LIN {X 0,Y 584.053,Z 357.982,A -85,B 0,C 180,E1 1855.602,E2 1855.602} C_VEL
LIN {X 0,Y 584.048,Z 357.978,A -85,B 0,C 180,E1 1852.272,E2 1852.272} C_VEL
LIN {X 0,Y 584.06,Z 357.981,A -85,B 0,C 180,E1 1849.289,E2 1849.289} C_VEL
LIN {X 0,Y 584.043,Z 357.976,A -85,B 0,C 180,E1 1845.968,E2 1845.968} C_VEL
LIN {X 0,Y 584.074,Z 357.982,A -85,B 0,C 180,E1 1842.948,E2 1842.948} C_VEL
LIN {X 0,Y 584.041,Z 357.978,A -85,B 0,C 180,E1 1839.765,E2 1839.765} C_VEL
LIN {X 0,Y 584.079,Z 357.983,A -85,B 0,C 180,E1 1836.687,E2 1836.687} C_VEL
LIN {X 0,Y 584.036,Z 357.983,A -85,B 0,C 180,E1 1833.454,E2 1833.454} C_VEL
LIN {X 0,Y 584.046,Z 358.076,A -85,B 0,C 180,E1 1833.218,E2 1833.218} C_VEL
LIN {X 0,Y 586.664,Z 365.487,A -85,B 0,C 180,E1 1832.47,E2 1832.47} C_VEL
LIN {X 0,Y 586.133,Z 402.245,A -85,B 0,C 180,E1 1829.65,E2 1829.65} C_VEL
LIN {X 0,Y 585.6,Z 444.184,A -85,B 0,C 180,E1 1826.531,E2 1826.531} C_VEL
LIN {X 0,Y 585.211,Z 489.388,A -85,B 0,C 180,E1 1823.299,E2 1823.299} C_VEL
LIN {X 0,Y 584.881,Z 536.224,A -85,B 0,C 180,E1 1820.024,E2 1820.024} C_VEL
LIN {X 0,Y 584.586,Z 583.959,A -85,B 0,C 180,E1 1816.75,E2 1816.75} C_VEL
LIN {X 0,Y 584.606,Z 588.885,A -85,B 0,C 180,E1 1816.44,E2 1816.44} C_VEL
LIN {X 0,Y 584.631,Z 729.653,A -85,B 0,C 180,E1 1814.662,E2 1814.662} C_VEL
LIN {X 0,Y 584.569,Z 745.603,A -85,B 0,C 180,E1 1814.307,E2 1814.307} C_VEL
LIN {X 0,Y 584.491,Z 761.576,A -85,B 0,C 180,E1 1813.756,E2 1813.756} C_VEL
LIN {X 0,Y 584.386,Z 776.468,A -85,B 0,C 180,E1 1813.053,E2 1813.053} C_VEL
LIN {X 0,Y 584.267,Z 791.891,A -85,B 0,C 180,E1 1812.094,E2 1812.094} C_VEL
LIN {X 0,Y 584.171,Z 804.549,A -85,B 0,C 180,E1 1811.093,E2 1811.093} C_VEL
LIN {X 0,Y 584.08,Z 817.071,A -85,B 0,C 180,E1 1809.857,E2 1809.857} C_VEL
LIN {X 0,Y 584.007,Z 827.449,A -85,B 0,C 180,E1 1808.566,E2 1808.566} C_VEL
LIN {X 0,Y 583.964,Z 836.343,A -85,B 0,C 180,E1 1807.18,E2 1807.18} C_VEL
LIN {X 0,Y 583.934,Z 843.646,A -85,B 0,C 180,E1 1805.7,E2 1805.7} C_VEL
LIN {X 0,Y 583.92,Z 849.058,A -85,B 0,C 180,E1 1804.223,E2 1804.223} C_VEL
LIN {X 0,Y 583.917,Z 852.97,A -85,B 0,C 180,E1 1802.65,E2 1802.65} C_VEL
LIN {X 0,Y 583.916,Z 855.029,A -85,B 0,C 180,E1 1801.08,E2 1801.08} C_VEL
LIN {X 0,Y 583.915,Z 855.387,A -85,B 0,C 180,E1 1799.412,E2 1799.412} C_VEL
LIN {X 0,Y 583.917,Z 853.911,A -85,B 0,C 180,E1 1797.841,E2 1797.841} C_VEL
LIN {X 0,Y 583.917,Z 850.708,A -85,B 0,C 180,E1 1796.269,E2 1796.269} C_VEL
LIN {X 0,Y 583.93,Z 845.646,A -85,B 0,C 180,E1 1794.695,E2 1794.695} C_VEL
LIN {X 0,Y 583.951,Z 838.942,A -85,B 0,C 180,E1 1793.215,E2 1793.215} C_VEL
LIN {X 0,Y 583.99,Z 830.831,A -85,B 0,C 180,E1 1791.831,E2 1791.831} C_VEL
LIN {X 0,Y 584.047,Z 821.249,A -85,B 0,C 180,E1 1790.541,E2 1790.541} C_VEL
LIN {X 0,Y 584.123,Z 810.24,A -85,B 0,C 180,E1 1789.347,E2 1789.347} C_VEL
LIN {X 0,Y 584.227,Z 797.718,A -85,B 0,C 180,E1 1788.249,E2 1788.249} C_VEL
LIN {X 0,Y 584.311,Z 784.011,A -85,B 0,C 180,E1 1787.298,E2 1787.298} C_VEL
LIN {X 0,Y 584.435,Z 769.379,A -85,B 0,C 180,E1 1786.496,E2 1786.496} C_VEL
LIN {X 0,Y 584.531,Z 754.061,A -85,B 0,C 180,E1 1785.872,E2 1785.872} C_VEL
LIN {X 0,Y 584.589,Z 738.598,A -85,B 0,C 180,E1 1785.426,E2 1785.426} C_VEL
LIN {X 0,Y 584.658,Z 721.58,A -85,B 0,C 180,E1 1785.13,E2 1785.13} C_VEL
LIN {X 0,Y 584.618,Z 588.986,A -85,B 0,C 180,E1 1783.472,E2 1783.472} C_VEL
LIN {X 0,Y 584.737,Z 556.999,A -85,B 0,C 180,E1 1781.317,E2 1781.317} C_VEL
LIN {X 0,Y 585.048,Z 511.693,A -85,B 0,C 180,E1 1778.179,E2 1778.179} C_VEL
LIN {X 0,Y 585.395,Z 465.881,A -85,B 0,C 180,E1 1774.939,E2 1774.939} C_VEL
LIN {X 0,Y 585.703,Z 443.805,A -85,B 0,C 180,E1 1773.323,E2 1773.323} C_VEL
LIN {X 0,Y 588.407,Z 405.449,A -85,B 0,C 180,E1 1770.07,E2 1770.07} C_VEL
LIN {X 0,Y 590.186,Z 385.24,A -85,B 0,C 180,E1 1768.262,E2 1768.262} C_VEL
LIN {X 0,Y 590.783,Z 371.274,A -85,B 0,C 180,E1 1766.805,E2 1766.805} C_VEL
LIN {X 0,Y 589.039,Z 367.53,A -85,B 0,C 180,E1 1766.051,E2 1766.051} C_VEL
LIN {X 0,Y 587.248,Z 364.067,A -85,B 0,C 180,E1 1765.224,E2 1765.224} C_VEL
LIN {X 0,Y 586.619,Z 362.881,A -85,B 0,C 180,E1 1764.899,E2 1764.899} C_VEL
LIN {X 0,Y 584.541,Z 359.787,A -85,B 0,C 180,E1 1763.673,E2 1763.673} C_VEL
LIN {X 0,Y 584.088,Z 358.254,A -85,B 0,C 180,E1 1762.7,E2 1762.7} C_VEL
LIN {X 0,Y 584.246,Z 358.829,A -85,B 0,C 180,E1 1761.928,E2 1761.928} C_VEL
LIN {X 0,Y 585.191,Z 361.195,A -85,B 0,C 180,E1 1761.167,E2 1761.167} C_VEL
LIN {X 0,Y 586.92,Z 363.366,A -85,B 0,C 180,E1 1760.612,E2 1760.612} C_VEL
LIN {X 0,Y 588.669,Z 367.246,A -85,B 0,C 180,E1 1760.057,E2 1760.057} C_VEL
LIN {X 0,Y 587.26,Z 390.715,A -85,B 0,C 180,E1 1758.655,E2 1758.655} C_VEL
LIN {X 0,Y 586.847,Z 427.382,A -85,B 0,C 180,E1 1756.679,E2 1756.679} C_VEL
LIN {X 0,Y 588.252,Z 442.511,A -85,B 0,C 180,E1 1755.823,E2 1755.823} C_VEL
LIN {X 0,Y 590.921,Z 453.438,A -85,B 0,C 180,E1 1755.124,E2 1755.124} C_VEL
LIN {X 0,Y 593.407,Z 459.109,A -85,B 0,C 180,E1 1754.68,E2 1754.68} C_VEL
LIN {X 0,Y 595.801,Z 462.899,A -85,B 0,C 180,E1 1754.227,E2 1754.227} C_VEL
LIN {X 0,Y 597.93,Z 465.232,A -85,B 0,C 180,E1 1753.748,E2 1753.748} C_VEL
LIN {X 0,Y 599.643,Z 466.302,A -85,B 0,C 180,E1 1753.226,E2 1753.226} C_VEL
LIN {X 0,Y 600.735,Z 465.901,A -85,B 0,C 180,E1 1752.637,E2 1752.637} C_VEL
LIN {X 0,Y 600.838,Z 464.09,A -85,B 0,C 180,E1 1752.117,E2 1752.117} C_VEL
LIN {X 0,Y 599.969,Z 460.825,A -85,B 0,C 180,E1 1751.63,E2 1751.63} C_VEL
LIN {X 0,Y 598.197,Z 456.293,A -85,B 0,C 180,E1 1751.238,E2 1751.238} C_VEL
LIN {X 0,Y 595.49,Z 449.308,A -85,B 0,C 180,E1 1750.915,E2 1750.915} C_VEL
LIN {X 0,Y 593.429,Z 440.344,A -85,B 0,C 180,E1 1750.685,E2 1750.685} C_VEL
LIN {X 0,Y 592.253,Z 428.653,A -85,B 0,C 180,E1 1750.553,E2 1750.553} C_VEL
LIN {X 0,Y 592.038,Z 404.531,A -85,B 0,C 180,E1 1750.528,E2 1750.528} C_VEL
LIN {X 0,Y 592.025,Z 368.885,A -85,B 0,C 180,E1 1750.527,E2 1750.527} C_VEL
LIN {X 0,Y 589.112,Z 365.245,A -85,B 0,C 180,E1 1750.194,E2 1750.194} C_VEL
LIN {X 0,Y 588.306,Z 364.085,A -85,B 0,C 180,E1 1750.101,E2 1750.101} C_VEL
LIN {X 0,Y 585.578,Z 361.73,A -85,B 0,C 180,E1 1749.783,E2 1749.783} C_VEL
LIN {X 0,Y 584.22,Z 358.714,A -85,B 0,C 180,E1 1749.623,E2 1749.623} C_VEL
LIN {X 0,Y 584.097,Z 357.981,A -85,B 0,C 180,E1 1749.585,E2 1749.585} C_VEL
LIN {X 0,Y 584.102,Z 357.996,A -85,B 0,C 180,E1 1749.495,E2 1749.495} C_VEL
LIN {X 0,Y 585.487,Z 361.592,A -85,B 0,C 180,E1 1749.167,E2 1749.167} C_VEL
LIN {X 0,Y 587.967,Z 367.026,A -85,B 0,C 180,E1 1748.647,E2 1748.647} C_VEL
LIN {X 0,Y 587.4,Z 418.925,A -85,B 0,C 180,E1 1745.668,E2 1745.668} C_VEL
LIN {X 0,Y 587.163,Z 455.345,A -85,B 0,C 180,E1 1743.661,E2 1743.661} C_VEL
LIN {X 0,Y 587.671,Z 460.738,A -85,B 0,C 180,E1 1743.55,E2 1743.55} C_VEL
LIN {X 0,Y 587.067,Z 677.552,A -85,B 0,C 180,E1 1740.523,E2 1740.523} C_VEL
LIN {X 0,Y 586.8,Z 761.949,A -85,B 0,C 180,E1 1739.34,E2 1739.34} C_VEL
LIN {X 0,Y 586.619,Z 783.698,A -85,B 0,C 180,E1 1738.843,E2 1738.843} C_VEL
LIN {X 0,Y 586.357,Z 806.115,A -85,B 0,C 180,E1 1738.137,E2 1738.137} C_VEL
LIN {X 0,Y 586.113,Z 827.151,A -85,B 0,C 180,E1 1737.28,E2 1737.28} C_VEL
LIN {X 0,Y 585.823,Z 846.743,A -85,B 0,C 180,E1 1736.29,E2 1736.29} C_VEL
LIN {X 0,Y 585.487,Z 867.144,A -85,B 0,C 180,E1 1735.057,E2 1735.057} C_VEL
LIN {X 0,Y 585.219,Z 885.801,A -85,B 0,C 180,E1 1733.726,E2 1733.726} C_VEL
LIN {X 0,Y 584.927,Z 904.1,A -85,B 0,C 180,E1 1732.196,E2 1732.196} C_VEL
LIN {X 0,Y 584.66,Z 921.221,A -85,B 0,C 180,E1 1730.523,E2 1730.523} C_VEL
LIN {X 0,Y 584.434,Z 936.724,A -85,B 0,C 180,E1 1728.762,E2 1728.762} C_VEL
LIN {X 0,Y 584.265,Z 950.748,A -85,B 0,C 180,E1 1726.914,E2 1726.914} C_VEL
LIN {X 0,Y 584.139,Z 963.342,A -85,B 0,C 180,E1 1724.979,E2 1724.979} C_VEL
LIN {X 0,Y 584.036,Z 974.372,A -85,B 0,C 180,E1 1722.96,E2 1722.96} C_VEL
LIN {X 0,Y 583.972,Z 983.482,A -85,B 0,C 180,E1 1720.956,E2 1720.956} C_VEL
LIN {X 0,Y 583.942,Z 991.15,A -85,B 0,C 180,E1 1718.897,E2 1718.897} C_VEL
LIN {X 0,Y 583.922,Z 997.17,A -85,B 0,C 180,E1 1716.786,E2 1716.786} C_VEL
LIN {X 0,Y 583.908,Z 1001.629,A -85,B 0,C 180,E1 1714.616,E2 1714.616} C_VEL
LIN {X 0,Y 583.897,Z 1004.326,A -85,B 0,C 180,E1 1712.552,E2 1712.552} C_VEL
LIN {X 0,Y 583.892,Z 1005.395,A -85,B 0,C 180,E1 1710.491,E2 1710.491} C_VEL
LIN {X 0,Y 583.899,Z 1004.954,A -85,B 0,C 180,E1 1708.332,E2 1708.332} C_VEL
LIN {X 0,Y 583.908,Z 1002.879,A -85,B 0,C 180,E1 1706.171,E2 1706.171} C_VEL
LIN {X 0,Y 583.918,Z 998.994,A -85,B 0,C 180,E1 1704.005,E2 1704.005} C_VEL
LIN {X 0,Y 583.937,Z 993.38,A -85,B 0,C 180,E1 1701.83,E2 1701.83} C_VEL
LIN {X 0,Y 583.97,Z 986.319,A -85,B 0,C 180,E1 1699.743,E2 1699.743} C_VEL
LIN {X 0,Y 584.013,Z 977.76,A -85,B 0,C 180,E1 1697.743,E2 1697.743} C_VEL
LIN {X 0,Y 584.102,Z 966.828,A -85,B 0,C 180,E1 1695.629,E2 1695.629} C_VEL
LIN {X 0,Y 584.228,Z 954.996,A -85,B 0,C 180,E1 1693.7,E2 1693.7} C_VEL
LIN {X 0,Y 584.377,Z 941.692,A -85,B 0,C 180,E1 1691.857,E2 1691.857} C_VEL
LIN {X 0,Y 584.559,Z 926.966,A -85,B 0,C 180,E1 1690.1,E2 1690.1} C_VEL
LIN {X 0,Y 584.807,Z 910.257,A -85,B 0,C 180,E1 1688.38,E2 1688.38} C_VEL
LIN {X 0,Y 585.104,Z 892.798,A -85,B 0,C 180,E1 1686.833,E2 1686.833} C_VEL
LIN {X 0,Y 585.409,Z 874.297,A -85,B 0,C 180,E1 1685.425,E2 1685.425} C_VEL
LIN {X 0,Y 585.679,Z 855.207,A -85,B 0,C 180,E1 1684.194,E2 1684.194} C_VEL
LIN {X 0,Y 585.986,Z 834.298,A -85,B 0,C 180,E1 1683.063,E2 1683.063} C_VEL
LIN {X 0,Y 586.307,Z 813.562,A -85,B 0,C 180,E1 1682.143,E2 1682.143} C_VEL
LIN {X 0,Y 586.515,Z 792.316,A -85,B 0,C 180,E1 1681.403,E2 1681.403} C_VEL
LIN {X 0,Y 586.726,Z 770.495,A -85,B 0,C 180,E1 1680.835,E2 1680.835} C_VEL
LIN {X 0,Y 586.869,Z 748.47,A -85,B 0,C 180,E1 1680.447,E2 1680.447} C_VEL
LIN {X 0,Y 587.486,Z 523.259,A -85,B 0,C 180,E1 1677.332,E2 1677.332} C_VEL
LIN {X 0,Y 587.485,Z 457.398,A -85,B 0,C 180,E1 1676.39,E2 1676.39} C_VEL
LIN {X 0,Y 587.058,Z 453.716,A -85,B 0,C 180,E1 1676.274,E2 1676.274} C_VEL
LIN {X 0,Y 587.62,Z 399.078,A -85,B 0,C 180,E1 1673.206,E2 1673.206} C_VEL
LIN {X 0,Y 587.877,Z 366.607,A -85,B 0,C 180,E1 1671.321,E2 1671.321} C_VEL
LIN {X 0,Y 584.335,Z 359.15,A -85,B 0,C 180,E1 1670.594,E2 1670.594} C_VEL
LIN {X 0,Y 584.1,Z 357.98,A -85,B 0,C 180,E1 1670.479,E2 1670.479} C_VEL
LIN {X 0,Y 584.117,Z 358.139,A -85,B 0,C 180,E1 1670.389,E2 1670.389} C_VEL
LIN {X 0,Y 585.254,Z 361.253,A -85,B 0,C 180,E1 1670.255,E2 1670.255} C_VEL
LIN {X 0,Y 587.659,Z 363.706,A -85,B 0,C 180,E1 1669.974,E2 1669.974} C_VEL
LIN {X 0,Y 588.786,Z 364.64,A -85,B 0,C 180,E1 1669.844,E2 1669.844} C_VEL
LIN {X 0,Y 591.535,Z 368.425,A -85,B 0,C 180,E1 1669.529,E2 1669.529} C_VEL
LIN {X 0,Y 592.035,Z 369.258,A -85,B 0,C 180,E1 1669.472,E2 1669.472} C_VEL
LIN {X 0,Y 592.224,Z 428.062,A -85,B 0,C 180,E1 1669.451,E2 1669.451} C_VEL
LIN {X 0,Y 593.343,Z 439.819,A -85,B 0,C 180,E1 1669.325,E2 1669.325} C_VEL
LIN {X 0,Y 595.364,Z 448.897,A -85,B 0,C 180,E1 1669.099,E2 1669.099} C_VEL
LIN {X 0,Y 598.058,Z 455.968,A -85,B 0,C 180,E1 1668.783,E2 1668.783} C_VEL
LIN {X 0,Y 599.889,Z 460.588,A -85,B 0,C 180,E1 1668.396,E2 1668.396} C_VEL
LIN {X 0,Y 600.807,Z 463.9,A -85,B 0,C 180,E1 1667.921,E2 1667.921} C_VEL
LIN {X 0,Y 600.841,Z 465.595,A -85,B 0,C 180,E1 1667.493,E2 1667.493} C_VEL
LIN {X 0,Y 600.174,Z 466.341,A -85,B 0,C 180,E1 1666.999,E2 1666.999} C_VEL
LIN {X 0,Y 598.675,Z 465.808,A -85,B 0,C 180,E1 1666.454,E2 1666.454} C_VEL
LIN {X 0,Y 596.53,Z 463.815,A -85,B 0,C 180,E1 1665.926,E2 1665.926} C_VEL
LIN {X 0,Y 593.903,Z 460.001,A -85,B 0,C 180,E1 1665.409,E2 1665.409} C_VEL
LIN {X 0,Y 591.267,Z 453.332,A -85,B 0,C 180,E1 1664.774,E2 1664.774} C_VEL
LIN {X 0,Y 589.42,Z 442.401,A -85,B 0,C 180,E1 1663.932,E2 1663.932} C_VEL
LIN {X 0,Y 589.031,Z 425.656,A -85,B 0,C 180,E1 1662.836,E2 1662.836} C_VEL
LIN {X 0,Y 589.555,Z 385.431,A -85,B 0,C 180,E1 1660.252,E2 1660.252} C_VEL
LIN {X 0,Y 589.749,Z 369.393,A -85,B 0,C 180,E1 1659.163,E2 1659.163} C_VEL
LIN {X 0,Y 586.078,Z 362.328,A -85,B 0,C 180,E1 1658.264,E2 1658.264} C_VEL
LIN {X 0,Y 584.273,Z 358.951,A -85,B 0,C 180,E1 1657.817,E2 1657.817} C_VEL
LIN {X 0,Y 584.093,Z 357.982,A -85,B 0,C 180,E1 1657.704,E2 1657.704} C_VEL
LIN {X 0,Y 584.07,Z 357.984,A -85,B 0,C 180,E1 1654.515,E2 1654.515} C_VEL
LIN {X 0,Y 584.087,Z 357.981,A -85,B 0,C 180,E1 1651.244,E2 1651.244} C_VEL
LIN {X 0,Y 584.097,Z 357.98,A -85,B 0,C 180,E1 1647.959,E2 1647.959} C_VEL
LIN {X 0,Y 584.087,Z 357.982,A -85,B 0,C 180,E1 1644.635,E2 1644.635} C_VEL
LIN {X 0,Y 584.1,Z 357.98,A -85,B 0,C 180,E1 1641.375,E2 1641.375} C_VEL
LIN {X 0,Y 584.098,Z 357.981,A -85,B 0,C 180,E1 1638.049,E2 1638.049} C_VEL
LIN {X 0,Y 584.092,Z 357.982,A -85,B 0,C 180,E1 1634.721,E2 1634.721} C_VEL
LIN {X 0,Y 584.1,Z 357.981,A -85,B 0,C 180,E1 1631.453,E2 1631.453} C_VEL
LIN {X 0,Y 584.092,Z 357.981,A -85,B 0,C 180,E1 1628.168,E2 1628.168} C_VEL
LIN {X 0,Y 584.084,Z 357.982,A -85,B 0,C 180,E1 1624.91,E2 1624.91} C_VEL
LIN {X 0,Y 584.095,Z 357.981,A -85,B 0,C 180,E1 1621.667,E2 1621.667} C_VEL
LIN {X 0,Y 584.084,Z 357.983,A -85,B 0,C 180,E1 1618.43,E2 1618.43} C_VEL
LIN {X 0,Y 584.099,Z 357.979,A -85,B 0,C 180,E1 1615.09,E2 1615.09} C_VEL
LIN {X 0,Y 584.079,Z 357.982,A -85,B 0,C 180,E1 1611.831,E2 1611.831} C_VEL
LIN {X 0,Y 584.092,Z 357.979,A -85,B 0,C 180,E1 1608.546,E2 1608.546} C_VEL
LIN {X 0,Y 584.096,Z 357.977,A -85,B 0,C 180,E1 1606.725,E2 1606.725} C_VEL
LIN {X 0,Y 583.11,Z 358.101,A -85,B 0,C 180,E1 1605.97,E2 1605.97} C_VEL
LIN {X 0,Y 576.657,Z 358.908,A -85,B 0,C 180,E1 1603.849,E2 1603.849} C_VEL
LIN {X 0,Y 576.112,Z 358.97,A -85,B 0,C 180,E1 1603.297,E2 1603.297} C_VEL
LIN {X 0,Y 576.132,Z 358.967,A -85,B 0,C 180,E1 1599.902,E2 1599.902} C_VEL
LIN {X 0,Y 576.129,Z 358.967,A -85,B 0,C 180,E1 1596.799,E2 1596.799} C_VEL
LIN {X 0,Y 576.111,Z 358.969,A -85,B 0,C 180,E1 1593.354,E2 1593.354} C_VEL
LIN {X 0,Y 576.151,Z 358.965,A -85,B 0,C 180,E1 1590.193,E2 1590.193} C_VEL
LIN {X 0,Y 576.105,Z 358.971,A -85,B 0,C 180,E1 1586.958,E2 1586.958} C_VEL
LIN {X 0,Y 576.154,Z 358.958,A -85,B 0,C 180,E1 1583.717,E2 1583.717} C_VEL
LIN {X 0,Y 576.109,Z 358.971,A -85,B 0,C 180,E1 1580.562,E2 1580.562} C_VEL
LIN {X 0,Y 576.137,Z 358.963,A -85,B 0,C 180,E1 1577.231,E2 1577.231} C_VEL
LIN {X 0,Y 576.126,Z 358.968,A -85,B 0,C 180,E1 1574.07,E2 1574.07} C_VEL
LIN {X 0,Y 576.115,Z 358.971,A -85,B 0,C 180,E1 1570.603,E2 1570.603} C_VEL
LIN {X 0,Y 576.151,Z 358.966,A -85,B 0,C 180,E1 1567.401,E2 1567.401} C_VEL
LIN {X 0,Y 576.105,Z 358.973,A -85,B 0,C 180,E1 1564.096,E2 1564.096} C_VEL
LIN {X 0,Y 576.174,Z 359.101,A -85,B 0,C 180,E1 1561.62,E2 1561.62} C_VEL
LIN {X 0,Y 578.943,Z 367.46,A -85,B 0,C 180,E1 1560.859,E2 1560.859} C_VEL
LIN {X 0,Y 578.406,Z 412.862,A -85,B 0,C 180,E1 1557.654,E2 1557.654} C_VEL
LIN {X 0,Y 577.861,Z 459.008,A -85,B 0,C 180,E1 1554.477,E2 1554.477} C_VEL
LIN {X 0,Y 577.806,Z 473.594,A -85,B 0,C 180,E1 1553.511,E2 1553.511} C_VEL
LIN {X 0,Y 578.38,Z 479.879,A -85,B 0,C 180,E1 1553.403,E2 1553.403} C_VEL
LIN {X 0,Y 577.837,Z 682.682,A -85,B 0,C 180,E1 1550.733,E2 1550.733} C_VEL
LIN {X 0,Y 577.692,Z 701.758,A -85,B 0,C 180,E1 1550.294,E2 1550.294} C_VEL
LIN {X 0,Y 577.499,Z 720.276,A -85,B 0,C 180,E1 1549.673,E2 1549.673} C_VEL
LIN {X 0,Y 577.252,Z 737.733,A -85,B 0,C 180,E1 1548.899,E2 1548.899} C_VEL
LIN {X 0,Y 577.042,Z 754.491,A -85,B 0,C 180,E1 1547.96,E2 1547.96} C_VEL
LIN {X 0,Y 576.794,Z 770.907,A -85,B 0,C 180,E1 1546.827,E2 1546.827} C_VEL
LIN {X 0,Y 576.56,Z 786.253,A -85,B 0,C 180,E1 1545.541,E2 1545.541} C_VEL
LIN {X 0,Y 576.357,Z 800.254,A -85,B 0,C 180,E1 1544.128,E2 1544.128} C_VEL
LIN {X 0,Y 576.205,Z 812.631,A -85,B 0,C 180,E1 1542.629,E2 1542.629} C_VEL
LIN {X 0,Y 576.087,Z 823.733,A -85,B 0,C 180,E1 1541.006,E2 1541.006} C_VEL
LIN {X 0,Y 575.998,Z 833.301,A -85,B 0,C 180,E1 1539.29,E2 1539.29} C_VEL
LIN {X 0,Y 575.956,Z 840.909,A -85,B 0,C 180,E1 1537.581,E2 1537.581} C_VEL
LIN {X 0,Y 575.92,Z 847.08,A -85,B 0,C 180,E1 1535.779,E2 1535.779} C_VEL
LIN {X 0,Y 575.919,Z 851.486,A -85,B 0,C 180,E1 1533.982,E2 1533.982} C_VEL
LIN {X 0,Y 575.917,Z 854.35,A -85,B 0,C 180,E1 1532.089,E2 1532.089} C_VEL
LIN {X 0,Y 575.911,Z 855.452,A -85,B 0,C 180,E1 1530.199,E2 1530.199} C_VEL
LIN {X 0,Y 575.913,Z 854.812,A -85,B 0,C 180,E1 1528.308,E2 1528.308} C_VEL
LIN {X 0,Y 575.909,Z 852.418,A -85,B 0,C 180,E1 1526.416,E2 1526.416} C_VEL
LIN {X 0,Y 575.923,Z 848.205,A -85,B 0,C 180,E1 1524.52,E2 1524.52} C_VEL
LIN {X 0,Y 575.941,Z 842.423,A -85,B 0,C 180,E1 1522.719,E2 1522.719} C_VEL
LIN {X 0,Y 575.998,Z 834.753,A -85,B 0,C 180,E1 1520.911,E2 1520.911} C_VEL
LIN {X 0,Y 576.07,Z 825.537,A -85,B 0,C 180,E1 1519.196,E2 1519.196} C_VEL
LIN {X 0,Y 576.188,Z 814.823,A -85,B 0,C 180,E1 1517.574,E2 1517.574} C_VEL
LIN {X 0,Y 576.334,Z 802.618,A -85,B 0,C 180,E1 1516.046,E2 1516.046} C_VEL
LIN {X 0,Y 576.522,Z 788.855,A -85,B 0,C 180,E1 1514.612,E2 1514.612} C_VEL
LIN {X 0,Y 576.747,Z 773.367,A -85,B 0,C 180,E1 1513.275,E2 1513.275} C_VEL
LIN {X 0,Y 576.986,Z 757.406,A -85,B 0,C 180,E1 1512.138,E2 1512.138} C_VEL
LIN {X 0,Y 577.194,Z 740.427,A -85,B 0,C 180,E1 1511.151,E2 1511.151} C_VEL
LIN {X 0,Y 577.461,Z 722.315,A -85,B 0,C 180,E1 1510.319,E2 1510.319} C_VEL
LIN {X 0,Y 577.664,Z 703.601,A -85,B 0,C 180,E1 1509.67,E2 1509.67} C_VEL
LIN {X 0,Y 577.822,Z 684.635,A -85,B 0,C 180,E1 1509.213,E2 1509.213} C_VEL
LIN {X 0,Y 577.938,Z 649.04,A -85,B 0,C 180,E1 1508.715,E2 1508.715} C_VEL
LIN {X 0,Y 578.207,Z 476.163,A -85,B 0,C 180,E1 1506.451,E2 1506.451} C_VEL
LIN {X 0,Y 577.737,Z 472.964,A -85,B 0,C 180,E1 1506.381,E2 1506.381} C_VEL
LIN {X 0,Y 578.229,Z 426.058,A -85,B 0,C 180,E1 1503.172,E2 1503.172} C_VEL
LIN {X 0,Y 578.809,Z 380.74,A -85,B 0,C 180,E1 1499.993,E2 1499.993} C_VEL
LIN {X 0,Y 578.729,Z 366.59,A -85,B 0,C 180,E1 1498.974,E2 1498.974} C_VEL
LIN {X 0,Y 576.1,Z 358.973,A -85,B 0,C 180,E1 1498.259,E2 1498.259} C_VEL
LIN {X 0,Y 576.155,Z 358.968,A -85,B 0,C 180,E1 1495.17,E2 1495.17} C_VEL
LIN {X 0,Y 576.096,Z 358.969,A -85,B 0,C 180,E1 1491.966,E2 1491.966} C_VEL
LIN {X 0,Y 576.163,Z 358.967,A -85,B 0,C 180,E1 1488.865,E2 1488.865} C_VEL
LIN {X 0,Y 576.096,Z 358.965,A -85,B 0,C 180,E1 1485.757,E2 1485.757} C_VEL
LIN {X 0,Y 576.16,Z 358.965,A -85,B 0,C 180,E1 1482.594,E2 1482.594} C_VEL
LIN {X 0,Y 576.095,Z 358.969,A -85,B 0,C 180,E1 1479.436,E2 1479.436} C_VEL
LIN {X 0,Y 576.157,Z 358.968,A -85,B 0,C 180,E1 1476.2,E2 1476.2} C_VEL
LIN {X 0,Y 576.127,Z 359.09,A -85,B 0,C 180,E1 1473.686,E2 1473.686} C_VEL
LIN {X 0,Y 579.582,Z 369.103,A -85,B 0,C 180,E1 1472.661,E2 1472.661} C_VEL
LIN {X 0,Y 579.005,Z 403.591,A -85,B 0,C 180,E1 1469.995,E2 1469.995} C_VEL
LIN {X 0,Y 578.244,Z 446.177,A -85,B 0,C 180,E1 1466.772,E2 1466.772} C_VEL
LIN {X 0,Y 577.665,Z 490.746,A -85,B 0,C 180,E1 1463.525,E2 1463.525} C_VEL
LIN {X 0,Y 577.219,Z 537.432,A -85,B 0,C 180,E1 1460.217,E2 1460.217} C_VEL
LIN {X 0,Y 576.827,Z 584.719,A -85,B 0,C 180,E1 1456.931,E2 1456.931} C_VEL
LIN {X 0,Y 576.855,Z 588.993,A -85,B 0,C 180,E1 1456.666,E2 1456.666} C_VEL
LIN {X 0,Y 577.147,Z 600.883,A -85,B 0,C 180,E1 1456.506,E2 1456.506} C_VEL
LIN {X 0,Y 576.881,Z 731.55,A -85,B 0,C 180,E1 1454.832,E2 1454.832} C_VEL
LIN {X 0,Y 576.789,Z 748.94,A -85,B 0,C 180,E1 1454.404,E2 1454.404} C_VEL
LIN {X 0,Y 576.665,Z 764.063,A -85,B 0,C 180,E1 1453.839,E2 1453.839} C_VEL
LIN {X 0,Y 576.528,Z 779.188,A -85,B 0,C 180,E1 1453.081,E2 1453.081} C_VEL
LIN {X 0,Y 576.379,Z 793.149,A -85,B 0,C 180,E1 1452.168,E2 1452.168} C_VEL
LIN {X 0,Y 576.252,Z 805.576,A -85,B 0,C 180,E1 1451.155,E2 1451.155} C_VEL
LIN {X 0,Y 576.127,Z 817.926,A -85,B 0,C 180,E1 1449.894,E2 1449.894} C_VEL
LIN {X 0,Y 576.042,Z 827.443,A -85,B 0,C 180,E1 1448.686,E2 1448.686} C_VEL
LIN {X 0,Y 575.983,Z 836.349,A -85,B 0,C 180,E1 1447.28,E2 1447.28} C_VEL
LIN {X 0,Y 575.941,Z 843.64,A -85,B 0,C 180,E1 1445.779,E2 1445.779} C_VEL
LIN {X 0,Y 575.922,Z 849.061,A -85,B 0,C 180,E1 1444.282,E2 1444.282} C_VEL
LIN {X 0,Y 575.917,Z 853.132,A -85,B 0,C 180,E1 1442.587,E2 1442.587} C_VEL
LIN {X 0,Y 575.916,Z 855.099,A -85,B 0,C 180,E1 1440.995,E2 1440.995} C_VEL
LIN {X 0,Y 575.913,Z 855.356,A -85,B 0,C 180,E1 1439.304,E2 1439.304} C_VEL
LIN {X 0,Y 575.916,Z 853.749,A -85,B 0,C 180,E1 1437.712,E2 1437.712} C_VEL
LIN {X 0,Y 575.918,Z 850.705,A -85,B 0,C 180,E1 1436.218,E2 1436.218} C_VEL
LIN {X 0,Y 575.934,Z 845.64,A -85,B 0,C 180,E1 1434.621,E2 1434.621} C_VEL
LIN {X 0,Y 575.963,Z 838.932,A -85,B 0,C 180,E1 1433.121,E2 1433.121} C_VEL
LIN {X 0,Y 576.023,Z 830.43,A -85,B 0,C 180,E1 1431.654,E2 1431.654} C_VEL
LIN {X 0,Y 576.101,Z 820.389,A -85,B 0,C 180,E1 1430.308,E2 1430.308} C_VEL
LIN {X 0,Y 576.215,Z 809.219,A -85,B 0,C 180,E1 1429.098,E2 1429.098} C_VEL
LIN {X 0,Y 576.346,Z 796.388,A -85,B 0,C 180,E1 1427.985,E2 1427.985} C_VEL
LIN {X 0,Y 576.473,Z 783.177,A -85,B 0,C 180,E1 1427.071,E2 1427.071} C_VEL
LIN {X 0,Y 576.623,Z 769.363,A -85,B 0,C 180,E1 1426.309,E2 1426.309} C_VEL
LIN {X 0,Y 576.75,Z 753.899,A -85,B 0,C 180,E1 1425.672,E2 1425.672} C_VEL
LIN {X 0,Y 576.835,Z 738.682,A -85,B 0,C 180,E1 1425.229,E2 1425.229} C_VEL
LIN {X 0,Y 576.926,Z 721.534,A -85,B 0,C 180,E1 1424.926,E2 1424.926} C_VEL
LIN {X 0,Y 576.936,Z 589.642,A -85,B 0,C 180,E1 1423.254,E2 1423.254} C_VEL
LIN {X 0,Y 576.795,Z 588.282,A -85,B 0,C 180,E1 1423.225,E2 1423.225} C_VEL
LIN {X 0,Y 577.176,Z 541.722,A -85,B 0,C 180,E1 1419.993,E2 1419.993} C_VEL
LIN {X 0,Y 577.596,Z 496.689,A -85,B 0,C 180,E1 1416.81,E2 1416.81} C_VEL
LIN {X 0,Y 577.991,Z 470.113,A -85,B 0,C 180,E1 1414.869,E2 1414.869} C_VEL
LIN {X 0,Y 580.438,Z 431.904,A -85,B 0,C 180,E1 1411.673,E2 1411.673} C_VEL
LIN {X 0,Y 583.743,Z 395.92,A -85,B 0,C 180,E1 1408.506,E2 1408.506} C_VEL
LIN {X 0,Y 584.535,Z 387.938,A -85,B 0,C 180,E1 1407.746,E2 1407.746} C_VEL
LIN {X 0,Y 585.228,Z 376.477,A -85,B 0,C 180,E1 1406.507,E2 1406.507} C_VEL
LIN {X 0,Y 584.104,Z 373.738,A -85,B 0,C 180,E1 1405.946,E2 1405.946} C_VEL
LIN {X 0,Y 582.291,Z 369.882,A -85,B 0,C 180,E1 1404.992,E2 1404.992} C_VEL
LIN {X 0,Y 580.184,Z 366.541,A -85,B 0,C 180,E1 1403.642,E2 1403.642} C_VEL
LIN {X 0,Y 579.927,Z 365.072,A -85,B 0,C 180,E1 1402.638,E2 1402.638} C_VEL
LIN {X 0,Y 580.077,Z 365.686,A -85,B 0,C 180,E1 1401.973,E2 1401.973} C_VEL
LIN {X 0,Y 581.144,Z 368.37,A -85,B 0,C 180,E1 1401.099,E2 1401.099} C_VEL
LIN {X 0,Y 581.997,Z 369.581,A -85,B 0,C 180,E1 1400.787,E2 1400.787} C_VEL
LIN {X 0,Y 582.794,Z 372.394,A -85,B 0,C 180,E1 1400.383,E2 1400.383} C_VEL
LIN {X 0,Y 580.924,Z 391.529,A -85,B 0,C 180,E1 1399.154,E2 1399.154} C_VEL
LIN {X 0,Y 579.746,Z 423.594,A -85,B 0,C 180,E1 1397.329,E2 1397.329} C_VEL
LIN {X 0,Y 580.76,Z 442.059,A -85,B 0,C 180,E1 1396.272,E2 1396.272} C_VEL
LIN {X 0,Y 583.215,Z 454.405,A -85,B 0,C 180,E1 1395.495,E2 1395.495} C_VEL
LIN {X 0,Y 586.437,Z 462.65,A -85,B 0,C 180,E1 1394.899,E2 1394.899} C_VEL
LIN {X 0,Y 590.275,Z 468.497,A -85,B 0,C 180,E1 1394.372,E2 1394.372} C_VEL
LIN {X 0,Y 593.495,Z 471.813,A -85,B 0,C 180,E1 1393.859,E2 1393.859} C_VEL
LIN {X 0,Y 596.154,Z 473.517,A -85,B 0,C 180,E1 1393.29,E2 1393.29} C_VEL
LIN {X 0,Y 597.785,Z 473.72,A -85,B 0,C 180,E1 1392.754,E2 1392.754} C_VEL
LIN {X 0,Y 598.567,Z 472.584,A -85,B 0,C 180,E1 1392.184,E2 1392.184} C_VEL
LIN {X 0,Y 598.237,Z 470.068,A -85,B 0,C 180,E1 1391.634,E2 1391.634} C_VEL
LIN {X 0,Y 596.756,Z 466.252,A -85,B 0,C 180,E1 1391.152,E2 1391.152} C_VEL
LIN {X 0,Y 594.306,Z 461.441,A -85,B 0,C 180,E1 1390.783,E2 1390.783} C_VEL
LIN {X 0,Y 591.051,Z 453.592,A -85,B 0,C 180,E1 1390.416,E2 1390.416} C_VEL
LIN {X 0,Y 588.688,Z 444.006,A -85,B 0,C 180,E1 1390.145,E2 1390.145} C_VEL
LIN {X 0,Y 587.281,Z 432.314,A -85,B 0,C 180,E1 1389.982,E2 1389.982} C_VEL
LIN {X 0,Y 586.874,Z 420.912,A -85,B 0,C 180,E1 1389.935,E2 1389.935} C_VEL
LIN {X 0,Y 586.779,Z 372.887,A -85,B 0,C 180,E1 1389.924,E2 1389.924} C_VEL
LIN {X 0,Y 584.938,Z 370.563,A -85,B 0,C 180,E1 1389.708,E2 1389.708} C_VEL
LIN {X 0,Y 582.868,Z 368.842,A -85,B 0,C 180,E1 1389.462,E2 1389.462} C_VEL
LIN {X 0,Y 580.966,Z 368.899,A -85,B 0,C 180,E1 1389.234,E2 1389.234} C_VEL
LIN {X 0,Y 580.371,Z 368.596,A -85,B 0,C 180,E1 1389.154,E2 1389.154} C_VEL
LIN {X 0,Y 581.351,Z 371.072,A -85,B 0,C 180,E1 1388.926,E2 1388.926} C_VEL
LIN {X 0,Y 580.582,Z 423.233,A -85,B 0,C 180,E1 1385.902,E2 1385.902} C_VEL
LIN {X 0,Y 580.273,Z 455.296,A -85,B 0,C 180,E1 1384.116,E2 1384.116} C_VEL
LIN {X 0,Y 580.995,Z 461.692,A -85,B 0,C 180,E1 1383.974,E2 1383.974} C_VEL
LIN {X 0,Y 580.173,Z 677.934,A -85,B 0,C 180,E1 1380.92,E2 1380.92} C_VEL
LIN {X 0,Y 579.818,Z 761.936,A -85,B 0,C 180,E1 1379.728,E2 1379.728} C_VEL
LIN {X 0,Y 579.571,Z 783.843,A -85,B 0,C 180,E1 1379.224,E2 1379.224} C_VEL
LIN {X 0,Y 579.234,Z 805.878,A -85,B 0,C 180,E1 1378.524,E2 1378.524} C_VEL
LIN {X 0,Y 578.901,Z 827.091,A -85,B 0,C 180,E1 1377.651,E2 1377.651} C_VEL
LIN {X 0,Y 578.501,Z 846.749,A -85,B 0,C 180,E1 1376.649,E2 1376.649} C_VEL
LIN {X 0,Y 578.067,Z 867.149,A -85,B 0,C 180,E1 1375.402,E2 1375.402} C_VEL
LIN {X 0,Y 577.691,Z 885.798,A -85,B 0,C 180,E1 1374.054,E2 1374.054} C_VEL
LIN {X 0,Y 577.292,Z 904.099,A -85,B 0,C 180,E1 1372.506,E2 1372.506} C_VEL
LIN {X 0,Y 576.927,Z 921.225,A -85,B 0,C 180,E1 1370.811,E2 1370.811} C_VEL
LIN {X 0,Y 576.632,Z 936.727,A -85,B 0,C 180,E1 1369.026,E2 1369.026} C_VEL
LIN {X 0,Y 576.394,Z 951.115,A -85,B 0,C 180,E1 1367.098,E2 1367.098} C_VEL
LIN {X 0,Y 576.227,Z 963.341,A -85,B 0,C 180,E1 1365.19,E2 1365.19} C_VEL
LIN {X 0,Y 576.086,Z 974.375,A -85,B 0,C 180,E1 1363.142,E2 1363.142} C_VEL
LIN {X 0,Y 575.999,Z 983.485,A -85,B 0,C 180,E1 1361.11,E2 1361.11} C_VEL
LIN {X 0,Y 575.955,Z 990.93,A -85,B 0,C 180,E1 1359.09,E2 1359.09} C_VEL
LIN {X 0,Y 575.916,Z 996.919,A -85,B 0,C 180,E1 1356.981,E2 1356.981} C_VEL
LIN {X 0,Y 575.902,Z 1001.507,A -85,B 0,C 180,E1 1354.76,E2 1354.76} C_VEL
LIN {X 0,Y 575.892,Z 1004.239,A -85,B 0,C 180,E1 1352.687,E2 1352.687} C_VEL
LIN {X 0,Y 575.892,Z 1005.373,A -85,B 0,C 180,E1 1350.597,E2 1350.597} C_VEL
LIN {X 0,Y 575.9,Z 1005.09,A -85,B 0,C 180,E1 1348.508,E2 1348.508} C_VEL
LIN {X 0,Y 575.908,Z 1003.122,A -85,B 0,C 180,E1 1346.317,E2 1346.317} C_VEL
LIN {X 0,Y 575.919,Z 999.408,A -85,B 0,C 180,E1 1344.121,E2 1344.121} C_VEL
LIN {X 0,Y 575.943,Z 994.292,A -85,B 0,C 180,E1 1342.017,E2 1342.017} C_VEL
LIN {X 0,Y 575.976,Z 987.411,A -85,B 0,C 180,E1 1339.902,E2 1339.902} C_VEL
LIN {X 0,Y 576.04,Z 978.688,A -85,B 0,C 180,E1 1337.775,E2 1337.775} C_VEL
LIN {X 0,Y 576.155,Z 968.568,A -85,B 0,C 180,E1 1335.734,E2 1335.734} C_VEL
LIN {X 0,Y 576.308,Z 956.994,A -85,B 0,C 180,E1 1333.78,E2 1333.78} C_VEL
LIN {X 0,Y 576.508,Z 943.777,A -85,B 0,C 180,E1 1331.881,E2 1331.881} C_VEL
LIN {X 0,Y 576.779,Z 928.359,A -85,B 0,C 180,E1 1329.978,E2 1329.978} C_VEL
LIN {X 0,Y 577.112,Z 911.918,A -85,B 0,C 180,E1 1328.238,E2 1328.238} C_VEL
LIN {X 0,Y 577.506,Z 894.393,A -85,B 0,C 180,E1 1326.642,E2 1326.642} C_VEL
LIN {X 0,Y 577.902,Z 875.757,A -85,B 0,C 180,E1 1325.193,E2 1325.193} C_VEL
LIN {X 0,Y 578.281,Z 856.995,A -85,B 0,C 180,E1 1323.949,E2 1323.949} C_VEL
LIN {X 0,Y 578.702,Z 836.642,A -85,B 0,C 180,E1 1322.813,E2 1322.813} C_VEL
LIN {X 0,Y 579.097,Z 816.267,A -85,B 0,C 180,E1 1321.878,E2 1321.878} C_VEL
LIN {X 0,Y 579.407,Z 794.841,A -85,B 0,C 180,E1 1321.102,E2 1321.102} C_VEL
LIN {X 0,Y 579.709,Z 772.624,A -85,B 0,C 180,E1 1320.493,E2 1320.493} C_VEL
LIN {X 0,Y 579.893,Z 750.519,A -85,B 0,C 180,E1 1320.086,E2 1320.086} C_VEL
LIN {X 0,Y 580.74,Z 525.93,A -85,B 0,C 180,E1 1316.943,E2 1316.943} C_VEL
LIN {X 0,Y 580.808,Z 458.677,A -85,B 0,C 180,E1 1315.97,E2 1315.97} C_VEL
LIN {X 0,Y 580.175,Z 453.716,A -85,B 0,C 180,E1 1315.819,E2 1315.819} C_VEL
LIN {X 0,Y 580.951,Z 398.315,A -85,B 0,C 180,E1 1312.668,E2 1312.668} C_VEL
LIN {X 0,Y 581.294,Z 370.395,A -85,B 0,C 180,E1 1311.029,E2 1311.029} C_VEL
LIN {X 0,Y 580.488,Z 368.645,A -85,B 0,C 180,E1 1310.824,E2 1310.824} C_VEL
LIN {X 0,Y 582.546,Z 368.956,A -85,B 0,C 180,E1 1310.576,E2 1310.576} C_VEL
LIN {X 0,Y 583.181,Z 368.938,A -85,B 0,C 180,E1 1310.5,E2 1310.5} C_VEL
LIN {X 0,Y 585.974,Z 371.724,A -85,B 0,C 180,E1 1310.17,E2 1310.17} C_VEL
LIN {X 0,Y 586.865,Z 373.003,A -85,B 0,C 180,E1 1310.066,E2 1310.066} C_VEL
LIN {X 0,Y 587.056,Z 428.35,A -85,B 0,C 180,E1 1310.044,E2 1310.044} C_VEL
LIN {X 0,Y 588.201,Z 441.017,A -85,B 0,C 180,E1 1309.911,E2 1309.911} C_VEL
LIN {X 0,Y 590.319,Z 451.175,A -85,B 0,C 180,E1 1309.667,E2 1309.667} C_VEL
LIN {X 0,Y 593.404,Z 459.611,A -85,B 0,C 180,E1 1309.318,E2 1309.318} C_VEL
LIN {X 0,Y 596.299,Z 465.318,A -85,B 0,C 180,E1 1308.938,E2 1308.938} C_VEL
LIN {X 0,Y 598.002,Z 469.329,A -85,B 0,C 180,E1 1308.482,E2 1308.482} C_VEL
LIN {X 0,Y 598.594,Z 472.122,A -85,B 0,C 180,E1 1307.948,E2 1307.948} C_VEL
LIN {X 0,Y 598.027,Z 473.599,A -85,B 0,C 180,E1 1307.362,E2 1307.362} C_VEL
LIN {X 0,Y 596.527,Z 473.66,A -85,B 0,C 180,E1 1306.812,E2 1306.812} C_VEL
LIN {X 0,Y 593.913,Z 472.146,A -85,B 0,C 180,E1 1306.218,E2 1306.218} C_VEL
LIN {X 0,Y 590.846,Z 469.178,A -85,B 0,C 180,E1 1305.71,E2 1305.71} C_VEL
LIN {X 0,Y 587.309,Z 463.738,A -85,B 0,C 180,E1 1305.089,E2 1305.089} C_VEL
LIN {X 0,Y 584.667,Z 455.987,A -85,B 0,C 180,E1 1304.371,E2 1304.371} C_VEL
LIN {X 0,Y 583.052,Z 444.678,A -85,B 0,C 180,E1 1303.499,E2 1303.499} C_VEL
LIN {X 0,Y 582.851,Z 425.123,A -85,B 0,C 180,E1 1302.218,E2 1302.218} C_VEL
LIN {X 0,Y 583.57,Z 385.886,A -85,B 0,C 180,E1 1299.659,E2 1299.659} C_VEL
LIN {X 0,Y 583.789,Z 373.683,A -85,B 0,C 180,E1 1298.818,E2 1298.818} C_VEL
LIN {X 0,Y 580.212,Z 367.32,A -85,B 0,C 180,E1 1297.966,E2 1297.966} C_VEL
LIN {X 0,Y 578.382,Z 363.585,A -85,B 0,C 180,E1 1297.481,E2 1297.481} C_VEL
LIN {X 0,Y 576.412,Z 360.302,A -85,B 0,C 180,E1 1297.007,E2 1297.007} C_VEL
LIN {X 0,Y 576.128,Z 358.973,A -85,B 0,C 180,E1 1296.865,E2 1296.865} C_VEL
LIN {X 0,Y 576.114,Z 358.965,A -85,B 0,C 180,E1 1293.497,E2 1293.497} C_VEL
LIN {X 0,Y 576.145,Z 358.967,A -85,B 0,C 180,E1 1290.332,E2 1290.332} C_VEL
LIN {X 0,Y 576.106,Z 358.971,A -85,B 0,C 180,E1 1287.046,E2 1287.046} C_VEL
LIN {X 0,Y 576.16,Z 358.964,A -85,B 0,C 180,E1 1283.85,E2 1283.85} C_VEL
LIN {X 0,Y 576.108,Z 358.97,A -85,B 0,C 180,E1 1280.629,E2 1280.629} C_VEL
LIN {X 0,Y 576.139,Z 358.966,A -85,B 0,C 180,E1 1277.263,E2 1277.263} C_VEL
LIN {X 0,Y 576.124,Z 358.968,A -85,B 0,C 180,E1 1274.164,E2 1274.164} C_VEL
LIN {X 0,Y 576.118,Z 358.97,A -85,B 0,C 180,E1 1270.798,E2 1270.798} C_VEL
LIN {X 0,Y 576.141,Z 358.967,A -85,B 0,C 180,E1 1267.679,E2 1267.679} C_VEL
LIN {X 0,Y 576.105,Z 358.971,A -85,B 0,C 180,E1 1264.28,E2 1264.28} C_VEL
LIN {X 0,Y 576.159,Z 358.965,A -85,B 0,C 180,E1 1261.094,E2 1261.094} C_VEL
LIN {X 0,Y 576.107,Z 358.972,A -85,B 0,C 180,E1 1257.911,E2 1257.911} C_VEL
LIN {X 0,Y 576.147,Z 358.966,A -85,B 0,C 180,E1 1254.622,E2 1254.622} C_VEL
LIN {X 0,Y 576.122,Z 358.97,A -85,B 0,C 180,E1 1251.416,E2 1251.416} C_VEL
LIN {X 0,Y 576.122,Z 358.969,A -85,B 0,C 180,E1 1248.081,E2 1248.081} C_VEL
LIN {X 0,Y 576.139,Z 358.966,A -85,B 0,C 180,E1 1244.911,E2 1244.911} C_VEL
LIN {X 0,Y 576.112,Z 358.97,A -85,B 0,C 180,E1 1243.297,E2 1243.297} C_VEL
LIN {X 0,Y 575.117,Z 359.099,A -85,B 0,C 180,E1 1242.531,E2 1242.531} C_VEL
LIN {X 0,Y 568.725,Z 359.894,A -85,B 0,C 180,E1 1240.38,E2 1240.38} C_VEL
LIN {X 0,Y 568.192,Z 359.956,A -85,B 0,C 180,E1 1239.82,E2 1239.82} C_VEL
LIN {X 0,Y 568.193,Z 359.956,A -85,B 0,C 180,E1 1236.675,E2 1236.675} C_VEL
LIN {X 0,Y 568.172,Z 359.958,A -85,B 0,C 180,E1 1233.337,E2 1233.337} C_VEL
LIN {X 0,Y 568.216,Z 359.953,A -85,B 0,C 180,E1 1230.133,E2 1230.133} C_VEL
LIN {X 0,Y 568.168,Z 359.96,A -85,B 0,C 180,E1 1226.818,E2 1226.818} C_VEL
LIN {X 0,Y 568.21,Z 359.946,A -85,B 0,C 180,E1 1223.504,E2 1223.504} C_VEL
LIN {X 0,Y 568.17,Z 359.96,A -85,B 0,C 180,E1 1220.424,E2 1220.424} C_VEL
LIN {X 0,Y 568.193,Z 359.952,A -85,B 0,C 180,E1 1217.058,E2 1217.058} C_VEL
LIN {X 0,Y 568.192,Z 359.956,A -85,B 0,C 180,E1 1213.894,E2 1213.894} C_VEL
LIN {X 0,Y 568.178,Z 359.961,A -85,B 0,C 180,E1 1210.493,E2 1210.493} C_VEL
LIN {X 0,Y 568.218,Z 359.955,A -85,B 0,C 180,E1 1207.251,E2 1207.251} C_VEL
LIN {X 0,Y 568.169,Z 359.962,A -85,B 0,C 180,E1 1204.017,E2 1204.017} C_VEL
LIN {X 0,Y 568.215,Z 360.061,A -85,B 0,C 180,E1 1202.009,E2 1202.009} C_VEL
LIN {X 0,Y 571.668,Z 370.395,A -85,B 0,C 180,E1 1201.061,E2 1201.061} C_VEL
LIN {X 0,Y 571.074,Z 413.667,A -85,B 0,C 180,E1 1197.984,E2 1197.984} C_VEL
LIN {X 0,Y 570.386,Z 459.793,A -85,B 0,C 180,E1 1194.765,E2 1194.765} C_VEL
LIN {X 0,Y 570.311,Z 473.64,A -85,B 0,C 180,E1 1193.839,E2 1193.839} C_VEL
LIN {X 0,Y 571.039,Z 480.443,A -85,B 0,C 180,E1 1193.715,E2 1193.715} C_VEL
LIN {X 0,Y 570.353,Z 682.696,A -85,B 0,C 180,E1 1191.018,E2 1191.018} C_VEL
LIN {X 0,Y 570.171,Z 701.769,A -85,B 0,C 180,E1 1190.574,E2 1190.574} C_VEL
LIN {X 0,Y 569.931,Z 720.164,A -85,B 0,C 180,E1 1189.951,E2 1189.951} C_VEL
LIN {X 0,Y 569.624,Z 737.75,A -85,B 0,C 180,E1 1189.162,E2 1189.162} C_VEL
LIN {X 0,Y 569.336,Z 755.029,A -85,B 0,C 180,E1 1188.177,E2 1188.177} C_VEL
LIN {X 0,Y 569.04,Z 770.918,A -85,B 0,C 180,E1 1187.063,E2 1187.063} C_VEL
LIN {X 0,Y 568.747,Z 786.118,A -85,B 0,C 180,E1 1185.774,E2 1185.774} C_VEL
LIN {X 0,Y 568.494,Z 799.991,A -85,B 0,C 180,E1 1184.358,E2 1184.358} C_VEL
LIN {X 0,Y 568.29,Z 812.64,A -85,B 0,C 180,E1 1182.808,E2 1182.808} C_VEL
LIN {X 0,Y 568.133,Z 823.734,A -85,B 0,C 180,E1 1181.162,E2 1181.162} C_VEL
LIN {X 0,Y 568.022,Z 833.302,A -85,B 0,C 180,E1 1179.422,E2 1179.422} C_VEL
LIN {X 0,Y 567.965,Z 841.1,A -85,B 0,C 180,E1 1177.64,E2 1177.64} C_VEL
LIN {X 0,Y 567.926,Z 847.082,A -85,B 0,C 180,E1 1175.86,E2 1175.86} C_VEL
LIN {X 0,Y 567.92,Z 851.487,A -85,B 0,C 180,E1 1174.038,E2 1174.038} C_VEL
LIN {X 0,Y 567.917,Z 854.351,A -85,B 0,C 180,E1 1172.119,E2 1172.119} C_VEL
LIN {X 0,Y 567.911,Z 855.452,A -85,B 0,C 180,E1 1170.201,E2 1170.201} C_VEL
LIN {X 0,Y 567.913,Z 854.811,A -85,B 0,C 180,E1 1168.285,E2 1168.285} C_VEL
LIN {X 0,Y 567.91,Z 852.417,A -85,B 0,C 180,E1 1166.366,E2 1166.366} C_VEL
LIN {X 0,Y 567.925,Z 848.204,A -85,B 0,C 180,E1 1164.443,E2 1164.443} C_VEL
LIN {X 0,Y 567.952,Z 842.422,A -85,B 0,C 180,E1 1162.616,E2 1162.616} C_VEL
LIN {X 0,Y 568.019,Z 834.752,A -85,B 0,C 180,E1 1160.782,E2 1160.782} C_VEL
LIN {X 0,Y 568.116,Z 825.532,A -85,B 0,C 180,E1 1159.043,E2 1159.043} C_VEL
LIN {X 0,Y 568.262,Z 814.815,A -85,B 0,C 180,E1 1157.398,E2 1157.398} C_VEL
LIN {X 0,Y 568.45,Z 802.609,A -85,B 0,C 180,E1 1155.848,E2 1155.848} C_VEL
LIN {X 0,Y 568.69,Z 788.846,A -85,B 0,C 180,E1 1154.395,E2 1154.395} C_VEL
LIN {X 0,Y 568.983,Z 773.36,A -85,B 0,C 180,E1 1153.039,E2 1153.039} C_VEL
LIN {X 0,Y 569.285,Z 757.4,A -85,B 0,C 180,E1 1151.888,E2 1151.888} C_VEL
LIN {X 0,Y 569.56,Z 740.421,A -85,B 0,C 180,E1 1150.889,E2 1150.889} C_VEL
LIN {X 0,Y 569.884,Z 722.309,A -85,B 0,C 180,E1 1150.047,E2 1150.047} C_VEL
LIN {X 0,Y 570.141,Z 703.592,A -85,B 0,C 180,E1 1149.39,E2 1149.39} C_VEL
LIN {X 0,Y 570.338,Z 684.462,A -85,B 0,C 180,E1 1148.924,E2 1148.924} C_VEL
LIN {X 0,Y 570.496,Z 644.488,A -85,B 0,C 180,E1 1148.364,E2 1148.364} C_VEL
LIN {X 0,Y 570.864,Z 477.218,A -85,B 0,C 180,E1 1146.144,E2 1146.144} C_VEL
LIN {X 0,Y 570.235,Z 472.954,A -85,B 0,C 180,E1 1146.051,E2 1146.051} C_VEL
LIN {X 0,Y 570.867,Z 426.048,A -85,B 0,C 180,E1 1142.797,E2 1142.797} C_VEL
LIN {X 0,Y 571.533,Z 382.145,A -85,B 0,C 180,E1 1139.687,E2 1139.687} C_VEL
LIN {X 0,Y 571.611,Z 369.861,A -85,B 0,C 180,E1 1138.8,E2 1138.8} C_VEL
LIN {X 0,Y 568.165,Z 359.964,A -85,B 0,C 180,E1 1137.863,E2 1137.863} C_VEL
LIN {X 0,Y 568.189,Z 359.957,A -85,B 0,C 180,E1 1134.564,E2 1134.564} C_VEL
LIN {X 0,Y 568.172,Z 359.96,A -85,B 0,C 180,E1 1131.467,E2 1131.467} C_VEL
LIN {X 0,Y 568.169,Z 359.956,A -85,B 0,C 180,E1 1128.107,E2 1128.107} C_VEL
LIN {X 0,Y 568.195,Z 359.955,A -85,B 0,C 180,E1 1125.024,E2 1125.024} C_VEL
LIN {X 0,Y 568.161,Z 359.954,A -85,B 0,C 180,E1 1121.74,E2 1121.74} C_VEL
LIN {X 0,Y 568.212,Z 359.955,A -85,B 0,C 180,E1 1118.621,E2 1118.621} C_VEL
LIN {X 0,Y 568.157,Z 359.961,A -85,B 0,C 180,E1 1115.379,E2 1115.379} C_VEL
LIN {X 0,Y 568.23,Z 360.016,A -85,B 0,C 180,E1 1114.177,E2 1114.177} C_VEL
LIN {X 0,Y 572.516,Z 372.196,A -85,B 0,C 180,E1 1112.898,E2 1112.898} C_VEL
LIN {X 0,Y 571.899,Z 404.937,A -85,B 0,C 180,E1 1110.349,E2 1110.349} C_VEL
LIN {X 0,Y 570.973,Z 447.521,A -85,B 0,C 180,E1 1107.084,E2 1107.084} C_VEL
LIN {X 0,Y 570.198,Z 489.454,A -85,B 0,C 180,E1 1103.956,E2 1103.956} C_VEL
LIN {X 0,Y 569.59,Z 536.691,A -85,B 0,C 180,E1 1100.554,E2 1100.554} C_VEL
LIN {X 0,Y 569.083,Z 584.728,A -85,B 0,C 180,E1 1097.168,E2 1097.168} C_VEL
LIN {X 0,Y 569.105,Z 589.023,A -85,B 0,C 180,E1 1096.9,E2 1096.9} C_VEL
LIN {X 0,Y 569.484,Z 597.5,A -85,B 0,C 180,E1 1096.779,E2 1096.779} C_VEL
LIN {X 0,Y 569.145,Z 731.336,A -85,B 0,C 180,E1 1095.041,E2 1095.041} C_VEL
LIN {X 0,Y 569.034,Z 748.162,A -85,B 0,C 180,E1 1094.631,E2 1094.631} C_VEL
LIN {X 0,Y 568.89,Z 762.75,A -85,B 0,C 180,E1 1094.089,E2 1094.089} C_VEL
LIN {X 0,Y 568.728,Z 776.457,A -85,B 0,C 180,E1 1093.419,E2 1093.419} C_VEL
LIN {X 0,Y 568.519,Z 791.774,A -85,B 0,C 180,E1 1092.442,E2 1092.442} C_VEL
LIN {X 0,Y 568.367,Z 803.842,A -85,B 0,C 180,E1 1091.466,E2 1091.466} C_VEL
LIN {X 0,Y 568.224,Z 815.248,A -85,B 0,C 180,E1 1090.34,E2 1090.34} C_VEL
LIN {X 0,Y 568.092,Z 825.99,A -85,B 0,C 180,E1 1089.012,E2 1089.012} C_VEL
LIN {X 0,Y 568.011,Z 834.695,A -85,B 0,C 180,E1 1087.674,E2 1087.674} C_VEL
LIN {X 0,Y 567.955,Z 842.809,A -85,B 0,C 180,E1 1086.064,E2 1086.064} C_VEL
LIN {X 0,Y 567.928,Z 848.429,A -85,B 0,C 180,E1 1084.544,E2 1084.544} C_VEL
LIN {X 0,Y 567.916,Z 852.575,A -85,B 0,C 180,E1 1082.927,E2 1082.927} C_VEL
LIN {X 0,Y 567.915,Z 854.857,A -85,B 0,C 180,E1 1081.312,E2 1081.312} C_VEL
LIN {X 0,Y 567.915,Z 855.454,A -85,B 0,C 180,E1 1079.698,E2 1079.698} C_VEL
LIN {X 0,Y 567.915,Z 854.212,A -85,B 0,C 180,E1 1077.982,E2 1077.982} C_VEL
LIN {X 0,Y 567.919,Z 851.191,A -85,B 0,C 180,E1 1076.366,E2 1076.366} C_VEL
LIN {X 0,Y 567.937,Z 846.383,A -85,B 0,C 180,E1 1074.748,E2 1074.748} C_VEL
LIN {X 0,Y 567.972,Z 839.937,A -85,B 0,C 180,E1 1073.227,E2 1073.227} C_VEL
LIN {X 0,Y 568.035,Z 832.098,A -85,B 0,C 180,E1 1071.803,E2 1071.803} C_VEL
LIN {X 0,Y 568.14,Z 822.071,A -85,B 0,C 180,E1 1070.376,E2 1070.376} C_VEL
LIN {X 0,Y 568.267,Z 811.214,A -85,B 0,C 180,E1 1069.149,E2 1069.149} C_VEL
LIN {X 0,Y 568.439,Z 798.976,A -85,B 0,C 180,E1 1068.021,E2 1068.021} C_VEL
LIN {X 0,Y 568.595,Z 785.585,A -85,B 0,C 180,E1 1067.044,E2 1067.044} C_VEL
LIN {X 0,Y 568.767,Z 772.318,A -85,B 0,C 180,E1 1066.272,E2 1066.272} C_VEL
LIN {X 0,Y 568.965,Z 756.816,A -85,B 0,C 180,E1 1065.576,E2 1065.576} C_VEL
LIN {X 0,Y 569.074,Z 741.27,A -85,B 0,C 180,E1 1065.09,E2 1065.09} C_VEL
LIN {X 0,Y 569.179,Z 725.781,A -85,B 0,C 180,E1 1064.776,E2 1064.776} C_VEL
LIN {X 0,Y 569.271,Z 590.432,A -85,B 0,C 180,E1 1063.033,E2 1063.033} C_VEL
LIN {X 0,Y 569.04,Z 588.272,A -85,B 0,C 180,E1 1062.989,E2 1062.989} C_VEL
LIN {X 0,Y 569.525,Z 541.713,A -85,B 0,C 180,E1 1059.713,E2 1059.713} C_VEL
LIN {X 0,Y 570.101,Z 499.279,A -85,B 0,C 180,E1 1056.649,E2 1056.649} C_VEL
LIN {X 0,Y 572.31,Z 461.026,A -85,B 0,C 180,E1 1053.489,E2 1053.489} C_VEL
LIN {X 0,Y 575.515,Z 421.656,A -85,B 0,C 180,E1 1050.092,E2 1050.092} C_VEL
LIN {X 0,Y 578.89,Z 392.925,A -85,B 0,C 180,E1 1047.446,E2 1047.446} C_VEL
LIN {X 0,Y 579.85,Z 381.79,A -85,B 0,C 180,E1 1046.216,E2 1046.216} C_VEL
LIN {X 0,Y 578.793,Z 379.377,A -85,B 0,C 180,E1 1045.664,E2 1045.664} C_VEL
LIN {X 0,Y 577.152,Z 375.646,A -85,B 0,C 180,E1 1044.647,E2 1044.647} C_VEL
LIN {X 0,Y 575.777,Z 372.966,A -85,B 0,C 180,E1 1043.443,E2 1043.443} C_VEL
LIN {X 0,Y 575.794,Z 371.905,A -85,B 0,C 180,E1 1042.521,E2 1042.521} C_VEL
LIN {X 0,Y 575.938,Z 373.055,A -85,B 0,C 180,E1 1041.828,E2 1041.828} C_VEL
LIN {X 0,Y 577.117,Z 375.493,A -85,B 0,C 180,E1 1041.031,E2 1041.031} C_VEL
LIN {X 0,Y 577.384,Z 376.975,A -85,B 0,C 180,E1 1040.797,E2 1040.797} C_VEL
LIN {X 0,Y 574.997,Z 392.706,A -85,B 0,C 180,E1 1039.695,E2 1039.695} C_VEL
LIN {X 0,Y 573.196,Z 418.004,A -85,B 0,C 180,E1 1038.146,E2 1038.146} C_VEL
LIN {X 0,Y 573.251,Z 438.242,A -85,B 0,C 180,E1 1036.955,E2 1036.955} C_VEL
LIN {X 0,Y 574.84,Z 451.603,A -85,B 0,C 180,E1 1036.121,E2 1036.121} C_VEL
LIN {X 0,Y 577.868,Z 462.537,A -85,B 0,C 180,E1 1035.374,E2 1035.374} C_VEL
LIN {X 0,Y 581.678,Z 470.16,A -85,B 0,C 180,E1 1034.772,E2 1034.772} C_VEL
LIN {X 0,Y 586.792,Z 476.492,A -85,B 0,C 180,E1 1034.164,E2 1034.164} C_VEL
LIN {X 0,Y 590.345,Z 479.419,A -85,B 0,C 180,E1 1033.681,E2 1033.681} C_VEL
LIN {X 0,Y 593.276,Z 480.949,A -85,B 0,C 180,E1 1033.136,E2 1033.136} C_VEL
LIN {X 0,Y 595.155,Z 481.133,A -85,B 0,C 180,E1 1032.613,E2 1032.613} C_VEL
LIN {X 0,Y 596.227,Z 479.999,A -85,B 0,C 180,E1 1031.999,E2 1031.999} C_VEL
LIN {X 0,Y 596.003,Z 477.531,A -85,B 0,C 180,E1 1031.42,E2 1031.42} C_VEL
LIN {X 0,Y 594.496,Z 473.93,A -85,B 0,C 180,E1 1030.911,E2 1030.911} C_VEL
LIN {X 0,Y 591.782,Z 469.212,A -85,B 0,C 180,E1 1030.499,E2 1030.499} C_VEL
LIN {X 0,Y 587.863,Z 461.173,A -85,B 0,C 180,E1 1030.05,E2 1030.05} C_VEL
LIN {X 0,Y 584.898,Z 451.667,A -85,B 0,C 180,E1 1029.703,E2 1029.703} C_VEL
LIN {X 0,Y 582.887,Z 440.383,A -85,B 0,C 180,E1 1029.464,E2 1029.464} C_VEL
LIN {X 0,Y 581.876,Z 426.578,A -85,B 0,C 180,E1 1029.343,E2 1029.343} C_VEL
LIN {X 0,Y 581.678,Z 379.945,A -85,B 0,C 180,E1 1029.319,E2 1029.319} C_VEL
LIN {X 0,Y 578.131,Z 386.209,A -85,B 0,C 180,E1 1028.888,E2 1028.888} C_VEL
LIN {X 0,Y 575.94,Z 388.306,A -85,B 0,C 180,E1 1028.617,E2 1028.617} C_VEL
LIN {X 0,Y 574.471,Z 388.296,A -85,B 0,C 180,E1 1028.431,E2 1028.431} C_VEL
LIN {X 0,Y 573.549,Z 438.993,A -85,B 0,C 180,E1 1025.487,E2 1025.487} C_VEL
LIN {X 0,Y 573.423,Z 455.311,A -85,B 0,C 180,E1 1024.58,E2 1024.58} C_VEL
LIN {X 0,Y 574.352,Z 462.862,A -85,B 0,C 180,E1 1024.404,E2 1024.404} C_VEL
LIN {X 0,Y 573.304,Z 678.825,A -85,B 0,C 180,E1 1021.319,E2 1021.319} C_VEL
LIN {X 0,Y 572.864,Z 761.923,A -85,B 0,C 180,E1 1020.126,E2 1020.126} C_VEL
LIN {X 0,Y 572.549,Z 784.042,A -85,B 0,C 180,E1 1019.613,E2 1019.613} C_VEL
LIN {X 0,Y 572.127,Z 806.447,A -85,B 0,C 180,E1 1018.89,E2 1018.89} C_VEL
LIN {X 0,Y 571.7,Z 827.684,A -85,B 0,C 180,E1 1018.002,E2 1018.002} C_VEL
LIN {X 0,Y 571.187,Z 847.751,A -85,B 0,C 180,E1 1016.961,E2 1016.961} C_VEL
LIN {X 0,Y 570.674,Z 867.155,A -85,B 0,C 180,E1 1015.755,E2 1015.755} C_VEL
LIN {X 0,Y 570.182,Z 885.796,A -85,B 0,C 180,E1 1014.392,E2 1014.392} C_VEL
LIN {X 0,Y 569.674,Z 904.098,A -85,B 0,C 180,E1 1012.823,E2 1012.823} C_VEL
LIN {X 0,Y 569.213,Z 921.229,A -85,B 0,C 180,E1 1011.106,E2 1011.106} C_VEL
LIN {X 0,Y 568.842,Z 936.731,A -85,B 0,C 180,E1 1009.296,E2 1009.296} C_VEL
LIN {X 0,Y 568.54,Z 950.755,A -85,B 0,C 180,E1 1007.396,E2 1007.396} C_VEL
LIN {X 0,Y 568.312,Z 963.406,A -85,B 0,C 180,E1 1005.395,E2 1005.395} C_VEL
LIN {X 0,Y 568.138,Z 974.377,A -85,B 0,C 180,E1 1003.329,E2 1003.329} C_VEL
LIN {X 0,Y 568.021,Z 983.896,A -85,B 0,C 180,E1 1001.165,E2 1001.165} C_VEL
LIN {X 0,Y 567.964,Z 991.562,A -85,B 0,C 180,E1 999.014,E2 999.014} C_VEL
LIN {X 0,Y 567.926,Z 997.43,A -85,B 0,C 180,E1 996.876,E2 996.876} C_VEL
LIN {X 0,Y 567.908,Z 1001.793,A -85,B 0,C 180,E1 994.646,E2 994.646} C_VEL
LIN {X 0,Y 567.898,Z 1004.4,A -85,B 0,C 180,E1 992.523,E2 992.523} C_VEL
LIN {X 0,Y 567.894,Z 1005.417,A -85,B 0,C 180,E1 990.404,E2 990.404} C_VEL
LIN {X 0,Y 567.903,Z 1004.891,A -85,B 0,C 180,E1 988.184,E2 988.184} C_VEL
LIN {X 0,Y 567.913,Z 1002.735,A -85,B 0,C 180,E1 985.962,E2 985.962} C_VEL
LIN {X 0,Y 567.928,Z 998.794,A -85,B 0,C 180,E1 983.734,E2 983.734} C_VEL
LIN {X 0,Y 567.949,Z 993.082,A -85,B 0,C 180,E1 981.496,E2 981.496} C_VEL
LIN {X 0,Y 568.007,Z 985.928,A -85,B 0,C 180,E1 979.349,E2 979.349} C_VEL
LIN {X 0,Y 568.105,Z 976.842,A -85,B 0,C 180,E1 977.188,E2 977.188} C_VEL
LIN {X 0,Y 568.255,Z 966.257,A -85,B 0,C 180,E1 975.115,E2 975.115} C_VEL
LIN {X 0,Y 568.476,Z 954.081,A -85,B 0,C 180,E1 973.098,E2 973.098} C_VEL
LIN {X 0,Y 568.774,Z 940.108,A -85,B 0,C 180,E1 971.128,E2 971.128} C_VEL
LIN {X 0,Y 569.146,Z 924.646,A -85,B 0,C 180,E1 969.269,E2 969.269} C_VEL
LIN {X 0,Y 569.561,Z 908.288,A -85,B 0,C 180,E1 967.577,E2 967.577} C_VEL
LIN {X 0,Y 570.048,Z 890.072,A -85,B 0,C 180,E1 965.956,E2 965.956} C_VEL
LIN {X 0,Y 570.563,Z 871.166,A -85,B 0,C 180,E1 964.519,E2 964.519} C_VEL
LIN {X 0,Y 571.121,Z 851.137,A -85,B 0,C 180,E1 963.233,E2 963.233} C_VEL
LIN {X 0,Y 571.586,Z 830.954,A -85,B 0,C 180,E1 962.157,E2 962.157} C_VEL
LIN {X 0,Y 572.074,Z 809.239,A -85,B 0,C 180,E1 961.216,E2 961.216} C_VEL
LIN {X 0,Y 572.509,Z 787.741,A -85,B 0,C 180,E1 960.491,E2 960.491} C_VEL
LIN {X 0,Y 572.786,Z 765.918,A -85,B 0,C 180,E1 959.951,E2 959.951} C_VEL
LIN {X 0,Y 573.048,Z 734.728,A -85,B 0,C 180,E1 959.465,E2 959.465} C_VEL
LIN {X 0,Y 574.153,Z 498.703,A -85,B 0,C 180,E1 956.113,E2 956.113} C_VEL
LIN {X 0,Y 574.157,Z 459.97,A -85,B 0,C 180,E1 955.539,E2 955.539} C_VEL
LIN {X 0,Y 573.316,Z 454.241,A -85,B 0,C 180,E1 955.382,E2 955.382} C_VEL
LIN {X 0,Y 574.289,Z 399.078,A -85,B 0,C 180,E1 952.205,E2 952.205} C_VEL
LIN {X 0,Y 574.535,Z 388.307,A -85,B 0,C 180,E1 951.559,E2 951.559} C_VEL
LIN {X 0,Y 576.248,Z 388.128,A -85,B 0,C 180,E1 951.344,E2 951.344} C_VEL
LIN {X 0,Y 578.913,Z 385.081,A -85,B 0,C 180,E1 951.016,E2 951.016} C_VEL
LIN {X 0,Y 581.763,Z 379.76,A -85,B 0,C 180,E1 950.67,E2 950.67} C_VEL
LIN {X 0,Y 581.961,Z 428.867,A -85,B 0,C 180,E1 950.646,E2 950.646} C_VEL
LIN {X 0,Y 583.122,Z 442.183,A -85,B 0,C 180,E1 950.508,E2 950.508} C_VEL
LIN {X 0,Y 585.254,Z 453.091,A -85,B 0,C 180,E1 950.255,E2 950.255} C_VEL
LIN {X 0,Y 588.382,Z 462.447,A -85,B 0,C 180,E1 949.89,E2 949.89} C_VEL
LIN {X 0,Y 592.419,Z 470.257,A -85,B 0,C 180,E1 949.427,E2 949.427} C_VEL
LIN {X 0,Y 594.937,Z 474.835,A -85,B 0,C 180,E1 948.984,E2 948.984} C_VEL
LIN {X 0,Y 596.148,Z 478.086,A -85,B 0,C 180,E1 948.475,E2 948.475} C_VEL
LIN {X 0,Y 596.212,Z 480.061,A -85,B 0,C 180,E1 947.98,E2 947.98} C_VEL
LIN {X 0,Y 595.135,Z 481.139,A -85,B 0,C 180,E1 947.38,E2 947.38} C_VEL
LIN {X 0,Y 592.837,Z 480.782,A -85,B 0,C 180,E1 946.768,E2 946.768} C_VEL
LIN {X 0,Y 589.795,Z 479.029,A -85,B 0,C 180,E1 946.235,E2 946.235} C_VEL
LIN {X 0,Y 585.177,Z 474.682,A -85,B 0,C 180,E1 945.578,E2 945.578} C_VEL
LIN {X 0,Y 581.197,Z 468.348,A -85,B 0,C 180,E1 944.857,E2 944.857} C_VEL
LIN {X 0,Y 578.441,Z 460.099,A -85,B 0,C 180,E1 944.086,E2 944.086} C_VEL
LIN {X 0,Y 576.743,Z 447.83,A -85,B 0,C 180,E1 943.126,E2 943.126} C_VEL
LIN {X 0,Y 576.631,Z 429.161,A -85,B 0,C 180,E1 941.88,E2 941.88} C_VEL
LIN {X 0,Y 577.546,Z 389.919,A -85,B 0,C 180,E1 939.299,E2 939.299} C_VEL
LIN {X 0,Y 577.871,Z 378.274,A -85,B 0,C 180,E1 938.495,E2 938.495} C_VEL
LIN {X 0,Y 572.525,Z 368.666,A -85,B 0,C 180,E1 937.175,E2 937.175} C_VEL
LIN {X 0,Y 570.271,Z 364.413,A -85,B 0,C 180,E1 936.581,E2 936.581} C_VEL
LIN {X 0,Y 568.448,Z 361.097,A -85,B 0,C 180,E1 936.103,E2 936.103} C_VEL
LIN {X 0,Y 568.221,Z 359.959,A -85,B 0,C 180,E1 935.96,E2 935.96} C_VEL
LIN {X 0,Y 568.219,Z 359.956,A -85,B 0,C 180,E1 932.578,E2 932.578} C_VEL
LIN {X 0,Y 568.205,Z 359.959,A -85,B 0,C 180,E1 929.215,E2 929.215} C_VEL
LIN {X 0,Y 568.22,Z 359.956,A -85,B 0,C 180,E1 925.873,E2 925.873} C_VEL
LIN {X 0,Y 568.2,Z 359.958,A -85,B 0,C 180,E1 922.557,E2 922.557} C_VEL
LIN {X 0,Y 568.186,Z 359.959,A -85,B 0,C 180,E1 919.319,E2 919.319} C_VEL
LIN {X 0,Y 568.211,Z 359.956,A -85,B 0,C 180,E1 916.101,E2 916.101} C_VEL
LIN {X 0,Y 568.185,Z 359.96,A -85,B 0,C 180,E1 912.81,E2 912.81} C_VEL
LIN {X 0,Y 568.219,Z 359.955,A -85,B 0,C 180,E1 909.521,E2 909.521} C_VEL
LIN {X 0,Y 568.18,Z 359.958,A -85,B 0,C 180,E1 906.162,E2 906.162} C_VEL
LIN {X 0,Y 568.2,Z 359.957,A -85,B 0,C 180,E1 902.824,E2 902.824} C_VEL
LIN {X 0,Y 568.194,Z 359.957,A -85,B 0,C 180,E1 899.596,E2 899.596} C_VEL
LIN {X 0,Y 568.17,Z 359.961,A -85,B 0,C 180,E1 896.165,E2 896.165} C_VEL
LIN {X 0,Y 568.214,Z 359.955,A -85,B 0,C 180,E1 892.951,E2 892.951} C_VEL
LIN {X 0,Y 568.167,Z 359.959,A -85,B 0,C 180,E1 889.648,E2 889.648} C_VEL
LIN {X 0,Y 568.212,Z 359.954,A -85,B 0,C 180,E1 886.361,E2 886.361} C_VEL
LIN {X 0,Y 568.172,Z 359.959,A -85,B 0,C 180,E1 883.2,E2 883.2} C_VEL
LIN {X 0,Y 568.192,Z 359.956,A -85,B 0,C 180,E1 879.82,E2 879.82} C_VEL
LIN {X 0,Y 567.192,Z 360.086,A -85,B 0,C 180,E1 879.043,E2 879.043} C_VEL
LIN {X 0,Y 560.776,Z 360.882,A -85,B 0,C 180,E1 876.862,E2 876.862} C_VEL
LIN {X 0,Y 560.276,Z 360.943,A -85,B 0,C 180,E1 876.294,E2 876.294} C_VEL
LIN {X 0,Y 560.251,Z 360.947,A -85,B 0,C 180,E1 872.929,E2 872.929} C_VEL
LIN {X 0,Y 560.279,Z 360.945,A -85,B 0,C 180,E1 869.666,E2 869.666} C_VEL
LIN {X 0,Y 560.25,Z 360.949,A -85,B 0,C 180,E1 866.41,E2 866.41} C_VEL
LIN {X 0,Y 560.275,Z 360.936,A -85,B 0,C 180,E1 863.029,E2 863.029} C_VEL
LIN {X 0,Y 560.282,Z 360.947,A -85,B 0,C 180,E1 859.641,E2 859.641} C_VEL
LIN {X 0,Y 560.279,Z 360.945,A -85,B 0,C 180,E1 856.282,E2 856.282} C_VEL
LIN {X 0,Y 560.263,Z 360.943,A -85,B 0,C 180,E1 852.971,E2 852.971} C_VEL
LIN {X 0,Y 560.282,Z 360.943,A -85,B 0,C 180,E1 849.708,E2 849.708} C_VEL
LIN {X 0,Y 560.254,Z 360.95,A -85,B 0,C 180,E1 846.335,E2 846.335} C_VEL
LIN {X 0,Y 560.273,Z 360.948,A -85,B 0,C 180,E1 842.99,E2 842.99} C_VEL
LIN {X 0,Y 560.268,Z 361.096,A -85,B 0,C 180,E1 842.422,E2 842.422} C_VEL
LIN {X 0,Y 564.455,Z 373.584,A -85,B 0,C 180,E1 841.266,E2 841.266} C_VEL
LIN {X 0,Y 563.761,Z 416.602,A -85,B 0,C 180,E1 838.181,E2 838.181} C_VEL
LIN {X 0,Y 562.9,Z 462.138,A -85,B 0,C 180,E1 834.952,E2 834.952} C_VEL
LIN {X 0,Y 562.828,Z 473.645,A -85,B 0,C 180,E1 834.177,E2 834.177} C_VEL
LIN {X 0,Y 563.712,Z 481.484,A -85,B 0,C 180,E1 834.029,E2 834.029} C_VEL
LIN {X 0,Y 562.886,Z 682.516,A -85,B 0,C 180,E1 831.314,E2 831.314} C_VEL
LIN {X 0,Y 562.667,Z 701.374,A -85,B 0,C 180,E1 830.872,E2 830.872} C_VEL
LIN {X 0,Y 562.374,Z 720.179,A -85,B 0,C 180,E1 830.231,E2 830.231} C_VEL
LIN {X 0,Y 562.011,Z 737.765,A -85,B 0,C 180,E1 829.432,E2 829.432} C_VEL
LIN {X 0,Y 561.665,Z 754.45,A -85,B 0,C 180,E1 828.473,E2 828.473} C_VEL
LIN {X 0,Y 561.294,Z 770.93,A -85,B 0,C 180,E1 827.306,E2 827.306} C_VEL
LIN {X 0,Y 560.937,Z 786.272,A -85,B 0,C 180,E1 825.985,E2 825.985} C_VEL
LIN {X 0,Y 560.635,Z 800,A -85,B 0,C 180,E1 824.564,E2 824.564} C_VEL
LIN {X 0,Y 560.382,Z 812.642,A -85,B 0,C 180,E1 822.992,E2 822.992} C_VEL
LIN {X 0,Y 560.184,Z 823.736,A -85,B 0,C 180,E1 821.323,E2 821.323} C_VEL
LIN {X 0,Y 560.05,Z 833.304,A -85,B 0,C 180,E1 819.557,E2 819.557} C_VEL
LIN {X 0,Y 559.974,Z 840.911,A -85,B 0,C 180,E1 817.799,E2 817.799} C_VEL
LIN {X 0,Y 559.932,Z 847.091,A -85,B 0,C 180,E1 815.942,E2 815.942} C_VEL
LIN {X 0,Y 559.921,Z 851.488,A -85,B 0,C 180,E1 814.096,E2 814.096} C_VEL
LIN {X 0,Y 559.916,Z 854.352,A -85,B 0,C 180,E1 812.149,E2 812.149} C_VEL
LIN {X 0,Y 559.911,Z 855.452,A -85,B 0,C 180,E1 810.204,E2 810.204} C_VEL
LIN {X 0,Y 559.913,Z 854.81,A -85,B 0,C 180,E1 808.26,E2 808.26} C_VEL
LIN {X 0,Y 559.912,Z 852.416,A -85,B 0,C 180,E1 806.314,E2 806.314} C_VEL
LIN {X 0,Y 559.926,Z 848.203,A -85,B 0,C 180,E1 804.363,E2 804.363} C_VEL
LIN {X 0,Y 559.963,Z 842.42,A -85,B 0,C 180,E1 802.51,E2 802.51} C_VEL
LIN {X 0,Y 560.041,Z 834.749,A -85,B 0,C 180,E1 800.65,E2 800.65} C_VEL
LIN {X 0,Y 560.164,Z 825.526,A -85,B 0,C 180,E1 798.885,E2 798.885} C_VEL
LIN {X 0,Y 560.342,Z 814.807,A -85,B 0,C 180,E1 797.217,E2 797.217} C_VEL
LIN {X 0,Y 560.572,Z 802.6,A -85,B 0,C 180,E1 795.645,E2 795.645} C_VEL
LIN {X 0,Y 560.872,Z 788.836,A -85,B 0,C 180,E1 794.172,E2 794.172} C_VEL
LIN {X 0,Y 561.23,Z 773.35,A -85,B 0,C 180,E1 792.798,E2 792.798} C_VEL
LIN {X 0,Y 561.605,Z 757.087,A -85,B 0,C 180,E1 791.611,E2 791.611} C_VEL
LIN {X 0,Y 561.939,Z 740.414,A -85,B 0,C 180,E1 790.619,E2 790.619} C_VEL
LIN {X 0,Y 562.317,Z 722.644,A -85,B 0,C 180,E1 789.781,E2 789.781} C_VEL
LIN {X 0,Y 562.624,Z 703.938,A -85,B 0,C 180,E1 789.113,E2 789.113} C_VEL
LIN {X 0,Y 562.863,Z 684.775,A -85,B 0,C 180,E1 788.637,E2 788.637} C_VEL
LIN {X 0,Y 563.04,Z 649.018,A -85,B 0,C 180,E1 788.124,E2 788.124} C_VEL
LIN {X 0,Y 563.535,Z 478.217,A -85,B 0,C 180,E1 785.828,E2 785.828} C_VEL
LIN {X 0,Y 562.751,Z 472.898,A -85,B 0,C 180,E1 785.709,E2 785.709} C_VEL
LIN {X 0,Y 563.546,Z 426.131,A -85,B 0,C 180,E1 782.414,E2 782.414} C_VEL
LIN {X 0,Y 564.338,Z 382.993,A -85,B 0,C 180,E1 779.318,E2 779.318} C_VEL
LIN {X 0,Y 564.34,Z 372.566,A -85,B 0,C 180,E1 778.559,E2 778.559} C_VEL
LIN {X 0,Y 560.257,Z 360.951,A -85,B 0,C 180,E1 777.447,E2 777.447} C_VEL
LIN {X 0,Y 560.223,Z 360.948,A -85,B 0,C 180,E1 774.124,E2 774.124} C_VEL
LIN {X 0,Y 560.286,Z 360.946,A -85,B 0,C 180,E1 770.922,E2 770.922} C_VEL
LIN {X 0,Y 560.22,Z 360.947,A -85,B 0,C 180,E1 767.712,E2 767.712} C_VEL
LIN {X 0,Y 560.275,Z 360.946,A -85,B 0,C 180,E1 764.452,E2 764.452} C_VEL
LIN {X 0,Y 560.224,Z 360.945,A -85,B 0,C 180,E1 761.289,E2 761.289} C_VEL
LIN {X 0,Y 560.241,Z 360.948,A -85,B 0,C 180,E1 757.923,E2 757.923} C_VEL
LIN {X 0,Y 560.241,Z 360.953,A -85,B 0,C 180,E1 754.818,E2 754.818} C_VEL
LIN {X 0,Y 560.263,Z 361.028,A -85,B 0,C 180,E1 754.684,E2 754.684} C_VEL
LIN {X 0,Y 565.482,Z 375.249,A -85,B 0,C 180,E1 753.148,E2 753.148} C_VEL
LIN {X 0,Y 564.683,Z 410.682,A -85,B 0,C 180,E1 750.366,E2 750.366} C_VEL
LIN {X 0,Y 563.682,Z 452.811,A -85,B 0,C 180,E1 747.121,E2 747.121} C_VEL
LIN {X 0,Y 562.777,Z 495.704,A -85,B 0,C 180,E1 743.896,E2 743.896} C_VEL
LIN {X 0,Y 561.964,Z 536.701,A -85,B 0,C 180,E1 740.846,E2 740.846} C_VEL
LIN {X 0,Y 561.337,Z 585.488,A -85,B 0,C 180,E1 737.359,E2 737.359} C_VEL
LIN {X 0,Y 561.362,Z 589.042,A -85,B 0,C 180,E1 737.141,E2 737.141} C_VEL
LIN {X 0,Y 561.827,Z 597.042,A -85,B 0,C 180,E1 737.021,E2 737.021} C_VEL
LIN {X 0,Y 561.417,Z 731.121,A -85,B 0,C 180,E1 735.257,E2 735.257} C_VEL
LIN {X 0,Y 561.288,Z 747.352,A -85,B 0,C 180,E1 734.864,E2 734.864} C_VEL
LIN {X 0,Y 561.124,Z 761.544,A -85,B 0,C 180,E1 734.341,E2 734.341} C_VEL
LIN {X 0,Y 560.927,Z 774.504,A -85,B 0,C 180,E1 733.714,E2 733.714} C_VEL
LIN {X 0,Y 560.724,Z 788.188,A -85,B 0,C 180,E1 732.879,E2 732.879} C_VEL
LIN {X 0,Y 560.507,Z 801.506,A -85,B 0,C 180,E1 731.838,E2 731.838} C_VEL
LIN {X 0,Y 560.323,Z 812.819,A -85,B 0,C 180,E1 730.747,E2 730.747} C_VEL
LIN {X 0,Y 560.171,Z 823.76,A -85,B 0,C 180,E1 729.452,E2 729.452} C_VEL
LIN {X 0,Y 560.053,Z 832.77,A -85,B 0,C 180,E1 728.108,E2 728.108} C_VEL
LIN {X 0,Y 559.982,Z 839.987,A -85,B 0,C 180,E1 726.768,E2 726.768} C_VEL
LIN {X 0,Y 559.941,Z 846.424,A -85,B 0,C 180,E1 725.225,E2 725.225} C_VEL
LIN {X 0,Y 559.92,Z 851.209,A -85,B 0,C 180,E1 723.584,E2 723.584} C_VEL
LIN {X 0,Y 559.916,Z 854.067,A -85,B 0,C 180,E1 722.047,E2 722.047} C_VEL
LIN {X 0,Y 559.914,Z 855.437,A -85,B 0,C 180,E1 720.307,E2 720.307} C_VEL
LIN {X 0,Y 559.915,Z 854.998,A -85,B 0,C 180,E1 718.772,E2 718.772} C_VEL
LIN {X 0,Y 559.916,Z 853.104,A -85,B 0,C 180,E1 717.237,E2 717.237} C_VEL
LIN {X 0,Y 559.928,Z 849.031,A -85,B 0,C 180,E1 715.494,E2 715.494} C_VEL
LIN {X 0,Y 559.953,Z 843.926,A -85,B 0,C 180,E1 714.039,E2 714.039} C_VEL
LIN {X 0,Y 560.017,Z 836.854,A -85,B 0,C 180,E1 712.511,E2 712.511} C_VEL
LIN {X 0,Y 560.11,Z 828.064,A -85,B 0,C 180,E1 711.066,E2 711.066} C_VEL
LIN {X 0,Y 560.235,Z 818.661,A -85,B 0,C 180,E1 709.823,E2 709.823} C_VEL
LIN {X 0,Y 560.424,Z 807.107,A -85,B 0,C 180,E1 708.578,E2 708.578} C_VEL
LIN {X 0,Y 560.612,Z 795.003,A -85,B 0,C 180,E1 707.538,E2 707.538} C_VEL
LIN {X 0,Y 560.798,Z 783.129,A -85,B 0,C 180,E1 706.703,E2 706.703} C_VEL
LIN {X 0,Y 561.019,Z 769.329,A -85,B 0,C 180,E1 705.921,E2 705.921} C_VEL
LIN {X 0,Y 561.208,Z 753.887,A -85,B 0,C 180,E1 705.269,E2 705.269} C_VEL
LIN {X 0,Y 561.342,Z 739.473,A -85,B 0,C 180,E1 704.835,E2 704.835} C_VEL
LIN {X 0,Y 561.475,Z 723.208,A -85,B 0,C 180,E1 704.524,E2 704.524} C_VEL
LIN {X 0,Y 561.615,Z 591.174,A -85,B 0,C 180,E1 702.805,E2 702.805} C_VEL
LIN {X 0,Y 561.296,Z 588.394,A -85,B 0,C 180,E1 702.757,E2 702.757} C_VEL
LIN {X 0,Y 561.902,Z 540.952,A -85,B 0,C 180,E1 699.371,E2 699.371} C_VEL
LIN {X 0,Y 562.231,Z 527.505,A -85,B 0,C 180,E1 698.346,E2 698.346} C_VEL
LIN {X 0,Y 564.27,Z 489.32,A -85,B 0,C 180,E1 695.225,E2 695.225} C_VEL
LIN {X 0,Y 567.221,Z 449.084,A -85,B 0,C 180,E1 691.808,E2 691.808} C_VEL
LIN {X 0,Y 570.84,Z 415.199,A -85,B 0,C 180,E1 688.771,E2 688.771} C_VEL
LIN {X 0,Y 573.46,Z 396.731,A -85,B 0,C 180,E1 686.998,E2 686.998} C_VEL
LIN {X 0,Y 574.524,Z 386.904,A -85,B 0,C 180,E1 685.864,E2 685.864} C_VEL
LIN {X 0,Y 572.6,Z 382.182,A -85,B 0,C 180,E1 684.569,E2 684.569} C_VEL
LIN {X 0,Y 571.476,Z 379.693,A -85,B 0,C 180,E1 683.372,E2 683.372} C_VEL
LIN {X 0,Y 571.65,Z 378.755,A -85,B 0,C 180,E1 682.506,E2 682.506} C_VEL
LIN {X 0,Y 571.788,Z 380.311,A -85,B 0,C 180,E1 681.735,E2 681.735} C_VEL
LIN {X 0,Y 572.433,Z 381.723,A -85,B 0,C 180,E1 681.252,E2 681.252} C_VEL
LIN {X 0,Y 569.419,Z 395.523,A -85,B 0,C 180,E1 680.195,E2 680.195} C_VEL
LIN {X 0,Y 567.102,Z 415.921,A -85,B 0,C 180,E1 678.838,E2 678.838} C_VEL
LIN {X 0,Y 566.357,Z 437.174,A -85,B 0,C 180,E1 677.525,E2 677.525} C_VEL
LIN {X 0,Y 567.471,Z 451.678,A -85,B 0,C 180,E1 676.594,E2 676.594} C_VEL
LIN {X 0,Y 570.228,Z 463.87,A -85,B 0,C 180,E1 675.744,E2 675.744} C_VEL
LIN {X 0,Y 574.007,Z 472.692,A -85,B 0,C 180,E1 675.063,E2 675.063} C_VEL
LIN {X 0,Y 578.596,Z 479.383,A -85,B 0,C 180,E1 674.464,E2 674.464} C_VEL
LIN {X 0,Y 584.07,Z 484.725,A -85,B 0,C 180,E1 673.888,E2 673.888} C_VEL
LIN {X 0,Y 587.938,Z 487.291,A -85,B 0,C 180,E1 673.398,E2 673.398} C_VEL
LIN {X 0,Y 590.987,Z 488.46,A -85,B 0,C 180,E1 672.854,E2 672.854} C_VEL
LIN {X 0,Y 593.088,Z 488.328,A -85,B 0,C 180,E1 672.261,E2 672.261} C_VEL
LIN {X 0,Y 593.997,Z 486.847,A -85,B 0,C 180,E1 671.637,E2 671.637} C_VEL
LIN {X 0,Y 593.543,Z 484.235,A -85,B 0,C 180,E1 671.07,E2 671.07} C_VEL
LIN {X 0,Y 591.701,Z 480.473,A -85,B 0,C 180,E1 670.553,E2 670.553} C_VEL
LIN {X 0,Y 588.064,Z 474.778,A -85,B 0,C 180,E1 670.073,E2 670.073} C_VEL
LIN {X 0,Y 583.822,Z 466.173,A -85,B 0,C 180,E1 669.576,E2 669.576} C_VEL
LIN {X 0,Y 580.571,Z 456.207,A -85,B 0,C 180,E1 669.186,E2 669.186} C_VEL
LIN {X 0,Y 578.287,Z 444.633,A -85,B 0,C 180,E1 668.908,E2 668.908} C_VEL
LIN {X 0,Y 577.014,Z 431.122,A -85,B 0,C 180,E1 668.751,E2 668.751} C_VEL
LIN {X 0,Y 576.733,Z 414.683,A -85,B 0,C 180,E1 668.716,E2 668.716} C_VEL
LIN {X 0,Y 576.682,Z 398.597,A -85,B 0,C 180,E1 668.709,E2 668.709} C_VEL
LIN {X 0,Y 572.756,Z 407.434,A -85,B 0,C 180,E1 668.217,E2 668.217} C_VEL
LIN {X 0,Y 569.753,Z 411.759,A -85,B 0,C 180,E1 667.832,E2 667.832} C_VEL
LIN {X 0,Y 568.223,Z 412.668,A -85,B 0,C 180,E1 667.633,E2 667.633} C_VEL
LIN {X 0,Y 567.391,Z 412.463,A -85,B 0,C 180,E1 667.522,E2 667.522} C_VEL
LIN {X 0,Y 566.61,Z 455.343,A -85,B 0,C 180,E1 665.056,E2 665.056} C_VEL
LIN {X 0,Y 567.741,Z 464.146,A -85,B 0,C 180,E1 664.843,E2 664.843} C_VEL
LIN {X 0,Y 566.462,Z 679.923,A -85,B 0,C 180,E1 661.725,E2 661.725} C_VEL
LIN {X 0,Y 565.937,Z 761.91,A -85,B 0,C 180,E1 660.534,E2 660.534} C_VEL
LIN {X 0,Y 565.554,Z 784.16,A -85,B 0,C 180,E1 660.014,E2 660.014} C_VEL
LIN {X 0,Y 565.045,Z 807.008,A -85,B 0,C 180,E1 659.265,E2 659.265} C_VEL
LIN {X 0,Y 564.539,Z 827.563,A -85,B 0,C 180,E1 658.395,E2 658.395} C_VEL
LIN {X 0,Y 563.914,Z 847.758,A -85,B 0,C 180,E1 657.337,E2 657.337} C_VEL
LIN {X 0,Y 563.286,Z 867.67,A -85,B 0,C 180,E1 656.082,E2 656.082} C_VEL
LIN {X 0,Y 562.667,Z 886.47,A -85,B 0,C 180,E1 654.683,E2 654.683} C_VEL
LIN {X 0,Y 562.043,Z 905.269,A -85,B 0,C 180,E1 653.04,E2 653.04} C_VEL
LIN {X 0,Y 561.476,Z 922.725,A -85,B 0,C 180,E1 651.247,E2 651.247} C_VEL
LIN {X 0,Y 561.018,Z 938.431,A -85,B 0,C 180,E1 649.36,E2 649.36} C_VEL
LIN {X 0,Y 560.654,Z 952.226,A -85,B 0,C 180,E1 647.426,E2 647.426} C_VEL
LIN {X 0,Y 560.382,Z 964.52,A -85,B 0,C 180,E1 645.418,E2 645.418} C_VEL
LIN {X 0,Y 560.18,Z 975.405,A -85,B 0,C 180,E1 643.312,E2 643.312} C_VEL
LIN {X 0,Y 560.04,Z 984.715,A -85,B 0,C 180,E1 641.117,E2 641.117} C_VEL
LIN {X 0,Y 559.961,Z 992.476,A -85,B 0,C 180,E1 638.834,E2 638.834} C_VEL
LIN {X 0,Y 559.935,Z 998.159,A -85,B 0,C 180,E1 636.666,E2 636.666} C_VEL
LIN {X 0,Y 559.919,Z 1002.271,A -85,B 0,C 180,E1 634.404,E2 634.404} C_VEL
LIN {X 0,Y 559.914,Z 1004.692,A -85,B 0,C 180,E1 632.149,E2 632.149} C_VEL
LIN {X 0,Y 559.909,Z 1005.489,A -85,B 0,C 180,E1 629.898,E2 629.898} C_VEL
LIN {X 0,Y 559.906,Z 1004.559,A -85,B 0,C 180,E1 627.646,E2 627.646} C_VEL
LIN {X 0,Y 559.911,Z 1001.954,A -85,B 0,C 180,E1 625.391,E2 625.391} C_VEL
LIN {X 0,Y 559.931,Z 997.703,A -85,B 0,C 180,E1 623.137,E2 623.137} C_VEL
LIN {X 0,Y 559.973,Z 991.87,A -85,B 0,C 180,E1 620.96,E2 620.96} C_VEL
LIN {X 0,Y 560.045,Z 984.31,A -85,B 0,C 180,E1 618.779,E2 618.779} C_VEL
LIN {X 0,Y 560.184,Z 974.955,A -85,B 0,C 180,E1 616.594,E2 616.594} C_VEL
LIN {X 0,Y 560.392,Z 963.876,A -85,B 0,C 180,E1 614.466,E2 614.466} C_VEL
LIN {X 0,Y 560.671,Z 951.47,A -85,B 0,C 180,E1 612.46,E2 612.46} C_VEL
LIN {X 0,Y 561.043,Z 937.469,A -85,B 0,C 180,E1 610.518,E2 610.518} C_VEL
LIN {X 0,Y 561.492,Z 922.233,A -85,B 0,C 180,E1 608.699,E2 608.699} C_VEL
LIN {X 0,Y 562.043,Z 905.276,A -85,B 0,C 180,E1 606.96,E2 606.96} C_VEL
LIN {X 0,Y 562.667,Z 886.478,A -85,B 0,C 180,E1 605.317,E2 605.317} C_VEL
LIN {X 0,Y 563.286,Z 867.671,A -85,B 0,C 180,E1 603.918,E2 603.918} C_VEL
LIN {X 0,Y 563.916,Z 847.718,A -85,B 0,C 180,E1 602.66,E2 602.66} C_VEL
LIN {X 0,Y 564.538,Z 827.575,A -85,B 0,C 180,E1 601.606,E2 601.606} C_VEL
LIN {X 0,Y 565.081,Z 805.923,A -85,B 0,C 180,E1 600.694,E2 600.694} C_VEL
LIN {X 0,Y 565.567,Z 782.862,A -85,B 0,C 180,E1 599.95,E2 599.95} C_VEL
LIN {X 0,Y 565.959,Z 760.62,A -85,B 0,C 180,E1 599.442,E2 599.442} C_VEL
LIN {X 0,Y 567.329,Z 532.216,A -85,B 0,C 180,E1 596.151,E2 596.151} C_VEL
LIN {X 0,Y 567.556,Z 461.357,A -85,B 0,C 180,E1 595.102,E2 595.102} C_VEL
LIN {X 0,Y 566.5,Z 454.241,A -85,B 0,C 180,E1 594.905,E2 594.905} C_VEL
LIN {X 0,Y 567.458,Z 412.489,A -85,B 0,C 180,E1 592.468,E2 592.468} C_VEL
LIN {X 0,Y 568.831,Z 412.459,A -85,B 0,C 180,E1 592.288,E2 592.288} C_VEL
LIN {X 0,Y 571.286,Z 409.87,A -85,B 0,C 180,E1 591.971,E2 591.971} C_VEL
LIN {X 0,Y 574.924,Z 402.958,A -85,B 0,C 180,E1 591.51,E2 591.51} C_VEL
LIN {X 0,Y 576.73,Z 398.469,A -85,B 0,C 180,E1 591.285,E2 591.285} C_VEL
LIN {X 0,Y 576.952,Z 429.837,A -85,B 0,C 180,E1 591.257,E2 591.257} C_VEL
LIN {X 0,Y 578.147,Z 443.617,A -85,B 0,C 180,E1 591.11,E2 591.11} C_VEL
LIN {X 0,Y 580.33,Z 455.26,A -85,B 0,C 180,E1 590.843,E2 590.843} C_VEL
LIN {X 0,Y 583.5,Z 465.36,A -85,B 0,C 180,E1 590.463,E2 590.463} C_VEL
LIN {X 0,Y 587.579,Z 473.95,A -85,B 0,C 180,E1 589.983,E2 589.983} C_VEL
LIN {X 0,Y 591.518,Z 480.16,A -85,B 0,C 180,E1 589.48,E2 589.48} C_VEL
LIN {X 0,Y 593.409,Z 483.884,A -85,B 0,C 180,E1 588.99,E2 588.99} C_VEL
LIN {X 0,Y 594.01,Z 486.63,A -85,B 0,C 180,E1 588.424,E2 588.424} C_VEL
LIN {X 0,Y 593.358,Z 488.155,A -85,B 0,C 180,E1 587.854,E2 587.854} C_VEL
LIN {X 0,Y 591.696,Z 488.565,A -85,B 0,C 180,E1 587.313,E2 587.313} C_VEL
LIN {X 0,Y 588.887,Z 487.757,A -85,B 0,C 180,E1 586.751,E2 586.751} C_VEL
LIN {X 0,Y 585.381,Z 485.707,A -85,B 0,C 180,E1 586.261,E2 586.261} C_VEL
LIN {X 0,Y 580.058,Z 480.841,A -85,B 0,C 180,E1 585.53,E2 585.53} C_VEL
LIN {X 0,Y 575.994,Z 474.779,A -85,B 0,C 180,E1 584.81,E2 584.81} C_VEL
LIN {X 0,Y 572.823,Z 466.565,A -85,B 0,C 180,E1 584.003,E2 584.003} C_VEL
LIN {X 0,Y 570.821,Z 455.408,A -85,B 0,C 180,E1 583.078,E2 583.078} C_VEL
LIN {X 0,Y 570.242,Z 441.021,A -85,B 0,C 180,E1 582.051,E2 582.051} C_VEL
LIN {X 0,Y 571.499,Z 395.41,A -85,B 0,C 180,E1 579.032,E2 579.032} C_VEL
LIN {X 0,Y 571.927,Z 382.983,A -85,B 0,C 180,E1 578.17,E2 578.17} C_VEL
LIN {X 0,Y 567.146,Z 374.212,A -85,B 0,C 180,E1 576.953,E2 576.953} C_VEL
LIN {X 0,Y 564.841,Z 369.989,A -85,B 0,C 180,E1 576.349,E2 576.349} C_VEL
LIN {X 0,Y 562.305,Z 365.37,A -85,B 0,C 180,E1 575.678,E2 575.678} C_VEL
LIN {X 0,Y 560.46,Z 362.104,A -85,B 0,C 180,E1 575.186,E2 575.186} C_VEL
LIN {X 0,Y 560.229,Z 360.952,A -85,B 0,C 180,E1 575.037,E2 575.037} C_VEL
LIN {X 0,Y 560.264,Z 360.947,A -85,B 0,C 180,E1 571.646,E2 571.646} C_VEL
LIN {X 0,Y 560.24,Z 360.948,A -85,B 0,C 180,E1 568.574,E2 568.574} C_VEL
LIN {X 0,Y 560.248,Z 360.947,A -85,B 0,C 180,E1 565.135,E2 565.135} C_VEL
LIN {X 0,Y 560.273,Z 360.943,A -85,B 0,C 180,E1 561.877,E2 561.877} C_VEL
LIN {X 0,Y 560.237,Z 360.948,A -85,B 0,C 180,E1 558.522,E2 558.522} C_VEL
LIN {X 0,Y 560.278,Z 360.942,A -85,B 0,C 180,E1 555.208,E2 555.208} C_VEL
LIN {X 0,Y 560.241,Z 360.949,A -85,B 0,C 180,E1 551.948,E2 551.948} C_VEL
LIN {X 0,Y 560.268,Z 360.947,A -85,B 0,C 180,E1 548.621,E2 548.621} C_VEL
LIN {X 0,Y 560.266,Z 360.946,A -85,B 0,C 180,E1 545.324,E2 545.324} C_VEL
LIN {X 0,Y 560.266,Z 360.949,A -85,B 0,C 180,E1 542.017,E2 542.017} C_VEL
LIN {X 0,Y 560.282,Z 360.947,A -85,B 0,C 180,E1 538.67,E2 538.67} C_VEL
LIN {X 0,Y 560.281,Z 360.947,A -85,B 0,C 180,E1 535.188,E2 535.188} C_VEL
LIN {X 0,Y 560.267,Z 360.949,A -85,B 0,C 180,E1 531.895,E2 531.895} C_VEL
LIN {X 0,Y 560.277,Z 360.947,A -85,B 0,C 180,E1 528.575,E2 528.575} C_VEL
LIN {X 0,Y 560.264,Z 360.945,A -85,B 0,C 180,E1 525.214,E2 525.214} C_VEL
LIN {X 0,Y 560.241,Z 360.948,A -85,B 0,C 180,E1 521.908,E2 521.908} C_VEL
LIN {X 0,Y 560.273,Z 360.944,A -85,B 0,C 180,E1 518.678,E2 518.678} C_VEL
LIN {X 0,Y 560.276,Z 360.943,A -85,B 0,C 180,E1 516.294,E2 516.294} C_VEL
LIN {X 0,Y 559.312,Z 361.068,A -85,B 0,C 180,E1 515.506,E2 515.506} C_VEL
LIN {X 0,Y 552.837,Z 361.873,A -85,B 0,C 180,E1 513.295,E2 513.295} C_VEL
LIN {X 0,Y 552.328,Z 361.935,A -85,B 0,C 180,E1 512.719,E2 512.719} C_VEL
LIN {X 0,Y 552.339,Z 361.935,A -85,B 0,C 180,E1 509.424,E2 509.424} C_VEL
LIN {X 0,Y 552.343,Z 361.933,A -85,B 0,C 180,E1 505.988,E2 505.988} C_VEL
LIN {X 0,Y 552.329,Z 361.929,A -85,B 0,C 180,E1 502.627,E2 502.627} C_VEL
LIN {X 0,Y 552.311,Z 361.935,A -85,B 0,C 180,E1 499.329,E2 499.329} C_VEL
LIN {X 0,Y 552.337,Z 361.936,A -85,B 0,C 180,E1 496.093,E2 496.093} C_VEL
LIN {X 0,Y 552.306,Z 361.932,A -85,B 0,C 180,E1 492.756,E2 492.756} C_VEL
LIN {X 0,Y 552.344,Z 361.928,A -85,B 0,C 180,E1 489.448,E2 489.448} C_VEL
LIN {X 0,Y 552.306,Z 361.939,A -85,B 0,C 180,E1 486.156,E2 486.156} C_VEL
LIN {X 0,Y 552.337,Z 362.027,A -85,B 0,C 180,E1 482.865,E2 482.865} C_VEL
LIN {X 0,Y 557.277,Z 375.926,A -85,B 0,C 180,E1 481.543,E2 481.543} C_VEL
LIN {X 0,Y 556.484,Z 419.79,A -85,B 0,C 180,E1 478.375,E2 478.375} C_VEL
LIN {X 0,Y 555.434,Z 463.737,A -85,B 0,C 180,E1 475.197,E2 475.197} C_VEL
LIN {X 0,Y 555.348,Z 473.563,A -85,B 0,C 180,E1 474.525,E2 474.525} C_VEL
LIN {X 0,Y 556.405,Z 482.412,A -85,B 0,C 180,E1 474.353,E2 474.353} C_VEL
LIN {X 0,Y 555.432,Z 682.53,A -85,B 0,C 180,E1 471.614,E2 471.614} C_VEL
LIN {X 0,Y 555.177,Z 701.262,A -85,B 0,C 180,E1 471.171,E2 471.171} C_VEL
LIN {X 0,Y 554.842,Z 719.438,A -85,B 0,C 180,E1 470.547,E2 470.547} C_VEL
LIN {X 0,Y 554.409,Z 737.779,A -85,B 0,C 180,E1 469.709,E2 469.709} C_VEL
LIN {X 0,Y 553.973,Z 755.267,A -85,B 0,C 180,E1 468.685,E2 468.685} C_VEL
LIN {X 0,Y 553.558,Z 770.941,A -85,B 0,C 180,E1 467.556,E2 467.556} C_VEL
LIN {X 0,Y 553.135,Z 786.282,A -85,B 0,C 180,E1 466.217,E2 466.217} C_VEL
LIN {X 0,Y 552.776,Z 800.008,A -85,B 0,C 180,E1 464.776,E2 464.776} C_VEL
LIN {X 0,Y 552.473,Z 812.674,A -85,B 0,C 180,E1 463.177,E2 463.177} C_VEL
LIN {X 0,Y 552.242,Z 823.737,A -85,B 0,C 180,E1 461.488,E2 461.488} C_VEL
LIN {X 0,Y 552.083,Z 833.305,A -85,B 0,C 180,E1 459.696,E2 459.696} C_VEL
LIN {X 0,Y 551.985,Z 840.913,A -85,B 0,C 180,E1 457.912,E2 457.912} C_VEL
LIN {X 0,Y 551.938,Z 847.205,A -85,B 0,C 180,E1 455.989,E2 455.989} C_VEL
LIN {X 0,Y 551.922,Z 851.694,A -85,B 0,C 180,E1 454.051,E2 454.051} C_VEL
LIN {X 0,Y 551.916,Z 854.465,A -85,B 0,C 180,E1 452.076,E2 452.076} C_VEL
LIN {X 0,Y 551.914,Z 855.474,A -85,B 0,C 180,E1 450.104,E2 450.104} C_VEL
LIN {X 0,Y 551.913,Z 854.743,A -85,B 0,C 180,E1 448.131,E2 448.131} C_VEL
LIN {X 0,Y 551.917,Z 852.257,A -85,B 0,C 180,E1 446.156,E2 446.156} C_VEL
LIN {X 0,Y 551.931,Z 847.937,A -85,B 0,C 180,E1 444.177,E2 444.177} C_VEL
LIN {X 0,Y 551.985,Z 841.823,A -85,B 0,C 180,E1 442.236,E2 442.236} C_VEL
LIN {X 0,Y 552.069,Z 834.244,A -85,B 0,C 180,E1 440.408,E2 440.408} C_VEL
LIN {X 0,Y 552.222,Z 824.893,A -85,B 0,C 180,E1 438.617,E2 438.617} C_VEL
LIN {X 0,Y 552.442,Z 814.04,A -85,B 0,C 180,E1 436.924,E2 436.924} C_VEL
LIN {X 0,Y 552.731,Z 801.68,A -85,B 0,C 180,E1 435.33,E2 435.33} C_VEL
LIN {X 0,Y 553.095,Z 787.736,A -85,B 0,C 180,E1 433.835,E2 433.835} C_VEL
LIN {X 0,Y 553.499,Z 772.929,A -85,B 0,C 180,E1 432.516,E2 432.516} C_VEL
LIN {X 0,Y 553.941,Z 756.584,A -85,B 0,C 180,E1 431.313,E2 431.313} C_VEL
LIN {X 0,Y 554.363,Z 739.413,A -85,B 0,C 180,E1 430.289,E2 430.289} C_VEL
LIN {X 0,Y 554.783,Z 722.079,A -85,B 0,C 180,E1 429.47,E2 429.47} C_VEL
LIN {X 0,Y 555.146,Z 703.285,A -85,B 0,C 180,E1 428.797,E2 428.797} C_VEL
LIN {X 0,Y 555.414,Z 684.225,A -85,B 0,C 180,E1 428.326,E2 428.326} C_VEL
LIN {X 0,Y 555.663,Z 638.148,A -85,B 0,C 180,E1 427.671,E2 427.671} C_VEL
LIN {X 0,Y 556.236,Z 479.351,A -85,B 0,C 180,E1 425.507,E2 425.507} C_VEL
LIN {X 0,Y 555.286,Z 472.831,A -85,B 0,C 180,E1 425.357,E2 425.357} C_VEL
LIN {X 0,Y 556.369,Z 425.807,A -85,B 0,C 180,E1 421.963,E2 421.963} C_VEL
LIN {X 0,Y 557.198,Z 381.442,A -85,B 0,C 180,E1 418.762,E2 418.762} C_VEL
LIN {X 0,Y 557.025,Z 375.301,A -85,B 0,C 180,E1 418.303,E2 418.303} C_VEL
LIN {X 0,Y 552.344,Z 361.937,A -85,B 0,C 180,E1 417.015,E2 417.015} C_VEL
LIN {X 0,Y 552.283,Z 361.938,A -85,B 0,C 180,E1 413.829,E2 413.829} C_VEL
LIN {X 0,Y 552.315,Z 361.933,A -85,B 0,C 180,E1 410.461,E2 410.461} C_VEL
LIN {X 0,Y 552.293,Z 361.937,A -85,B 0,C 180,E1 407.384,E2 407.384} C_VEL
LIN {X 0,Y 552.295,Z 361.936,A -85,B 0,C 180,E1 404.042,E2 404.042} C_VEL
LIN {X 0,Y 552.323,Z 361.935,A -85,B 0,C 180,E1 400.826,E2 400.826} C_VEL
LIN {X 0,Y 552.282,Z 361.939,A -85,B 0,C 180,E1 397.536,E2 397.536} C_VEL
LIN {X 0,Y 552.29,Z 362.014,A -85,B 0,C 180,E1 395.213,E2 395.213} C_VEL
LIN {X 0,Y 558.483,Z 378.318,A -85,B 0,C 180,E1 393.409,E2 393.409} C_VEL
LIN {X 0,Y 557.565,Z 414.371,A -85,B 0,C 180,E1 390.557,E2 390.557} C_VEL
LIN {X 0,Y 556.427,Z 456.628,A -85,B 0,C 180,E1 387.272,E2 387.272} C_VEL
LIN {X 0,Y 555.392,Z 500.436,A -85,B 0,C 180,E1 383.952,E2 383.952} C_VEL
LIN {X 0,Y 554.275,Z 544.954,A -85,B 0,C 180,E1 380.572,E2 380.572} C_VEL
LIN {X 0,Y 553.563,Z 588.447,A -85,B 0,C 180,E1 377.399,E2 377.399} C_VEL
LIN {X 0,Y 554.181,Z 597.093,A -85,B 0,C 180,E1 377.264,E2 377.264} C_VEL
LIN {X 0,Y 553.699,Z 730.715,A -85,B 0,C 180,E1 375.481,E2 375.481} C_VEL
LIN {X 0,Y 553.547,Z 747.024,A -85,B 0,C 180,E1 375.088,E2 375.088} C_VEL
LIN {X 0,Y 553.349,Z 761.534,A -85,B 0,C 180,E1 374.547,E2 374.547} C_VEL
LIN {X 0,Y 553.119,Z 774.498,A -85,B 0,C 180,E1 373.912,E2 373.912} C_VEL
LIN {X 0,Y 552.878,Z 788.193,A -85,B 0,C 180,E1 373.065,E2 373.065} C_VEL
LIN {X 0,Y 552.623,Z 801.5,A -85,B 0,C 180,E1 372.01,E2 372.01} C_VEL
LIN {X 0,Y 552.416,Z 812.316,A -85,B 0,C 180,E1 370.956,E2 370.956} C_VEL
LIN {X 0,Y 552.236,Z 822.993,A -85,B 0,C 180,E1 369.694,E2 369.694} C_VEL
LIN {X 0,Y 552.082,Z 832.764,A -85,B 0,C 180,E1 368.226,E2 368.226} C_VEL
LIN {X 0,Y 551.996,Z 839.982,A -85,B 0,C 180,E1 366.866,E2 366.866} C_VEL
LIN {X 0,Y 551.946,Z 846.429,A -85,B 0,C 180,E1 365.301,E2 365.301} C_VEL
LIN {X 0,Y 551.921,Z 850.963,A -85,B 0,C 180,E1 363.74,E2 363.74} C_VEL
LIN {X 0,Y 551.915,Z 853.748,A -85,B 0,C 180,E1 362.284,E2 362.284} C_VEL
LIN {X 0,Y 551.915,Z 855.36,A -85,B 0,C 180,E1 360.623,E2 360.623} C_VEL
LIN {X 0,Y 551.916,Z 855.146,A -85,B 0,C 180,E1 358.962,E2 358.962} C_VEL
LIN {X 0,Y 551.915,Z 853.412,A -85,B 0,C 180,E1 357.404,E2 357.404} C_VEL
LIN {X 0,Y 551.929,Z 849.931,A -85,B 0,C 180,E1 355.741,E2 355.741} C_VEL
LIN {X 0,Y 551.956,Z 844.809,A -85,B 0,C 180,E1 354.178,E2 354.178} C_VEL
LIN {X 0,Y 552.016,Z 838.391,A -85,B 0,C 180,E1 352.716,E2 352.716} C_VEL
LIN {X 0,Y 552.124,Z 830.174,A -85,B 0,C 180,E1 351.251,E2 351.251} C_VEL
LIN {X 0,Y 552.27,Z 820.348,A -85,B 0,C 180,E1 349.886,E2 349.886} C_VEL
LIN {X 0,Y 552.456,Z 810.183,A -85,B 0,C 180,E1 348.729,E2 348.729} C_VEL
LIN {X 0,Y 552.704,Z 797.686,A -85,B 0,C 180,E1 347.569,E2 347.569} C_VEL
LIN {X 0,Y 552.935,Z 784.726,A -85,B 0,C 180,E1 346.617,E2 346.617} C_VEL
LIN {X 0,Y 553.163,Z 772.257,A -85,B 0,C 180,E1 345.877,E2 345.877} C_VEL
LIN {X 0,Y 553.428,Z 757.334,A -85,B 0,C 180,E1 345.183,E2 345.183} C_VEL
LIN {X 0,Y 553.592,Z 741.719,A -85,B 0,C 180,E1 344.677,E2 344.677} C_VEL
LIN {X 0,Y 553.724,Z 727.642,A -85,B 0,C 180,E1 344.376,E2 344.376} C_VEL
LIN {X 0,Y 553.973,Z 591.989,A -85,B 0,C 180,E1 342.572,E2 342.572} C_VEL
LIN {X 0,Y 553.564,Z 588.206,A -85,B 0,C 180,E1 342.495,E2 342.495} C_VEL
LIN {X 0,Y 553.969,Z 565.456,A -85,B 0,C 180,E1 340.823,E2 340.823} C_VEL
LIN {X 0,Y 555.954,Z 522.583,A -85,B 0,C 180,E1 337.365,E2 337.365} C_VEL
LIN {X 0,Y 558.704,Z 480.832,A -85,B 0,C 180,E1 333.881,E2 333.881} C_VEL
LIN {X 0,Y 561.838,Z 445.191,A -85,B 0,C 180,E1 330.758,E2 330.758} C_VEL
LIN {X 0,Y 566.079,Z 412.945,A -85,B 0,C 180,E1 327.764,E2 327.764} C_VEL
LIN {X 0,Y 568.285,Z 400.01,A -85,B 0,C 180,E1 326.464,E2 326.464} C_VEL
LIN {X 0,Y 569.447,Z 392.421,A -85,B 0,C 180,E1 325.572,E2 325.572} C_VEL
LIN {X 0,Y 567.87,Z 388.469,A -85,B 0,C 180,E1 324.353,E2 324.353} C_VEL
LIN {X 0,Y 567.219,Z 386.189,A -85,B 0,C 180,E1 323.158,E2 323.158} C_VEL
LIN {X 0,Y 567.504,Z 385.656,A -85,B 0,C 180,E1 322.44,E2 322.44} C_VEL
LIN {X 0,Y 567.539,Z 387.821,A -85,B 0,C 180,E1 321.627,E2 321.627} C_VEL
LIN {X 0,Y 563.966,Z 400.342,A -85,B 0,C 180,E1 320.603,E2 320.603} C_VEL
LIN {X 0,Y 561.215,Z 417.526,A -85,B 0,C 180,E1 319.373,E2 319.373} C_VEL
LIN {X 0,Y 559.831,Z 437.06,A -85,B 0,C 180,E1 318.09,E2 318.09} C_VEL
LIN {X 0,Y 560.557,Z 453.372,A -85,B 0,C 180,E1 316.997,E2 316.997} C_VEL
LIN {X 0,Y 562.998,Z 465.928,A -85,B 0,C 180,E1 316.092,E2 316.092} C_VEL
LIN {X 0,Y 566.444,Z 475.087,A -85,B 0,C 180,E1 315.37,E2 315.37} C_VEL
LIN {X 0,Y 571.088,Z 482.75,A -85,B 0,C 180,E1 314.699,E2 314.699} C_VEL
LIN {X 0,Y 577.121,Z 489.335,A -85,B 0,C 180,E1 314.03,E2 314.03} C_VEL
LIN {X 0,Y 582.802,Z 493.56,A -85,B 0,C 180,E1 313.473,E2 313.473} C_VEL
LIN {X 0,Y 586.424,Z 495.331,A -85,B 0,C 180,E1 312.992,E2 312.992} C_VEL
LIN {X 0,Y 589.326,Z 495.928,A -85,B 0,C 180,E1 312.437,E2 312.437} C_VEL
LIN {X 0,Y 591.046,Z 495.414,A -85,B 0,C 180,E1 311.898,E2 311.898} C_VEL
LIN {X 0,Y 591.738,Z 493.705,A -85,B 0,C 180,E1 311.287,E2 311.287} C_VEL
LIN {X 0,Y 591.018,Z 490.845,A -85,B 0,C 180,E1 310.706,E2 310.706} C_VEL
LIN {X 0,Y 588.935,Z 487.112,A -85,B 0,C 180,E1 310.209,E2 310.209} C_VEL
LIN {X 0,Y 583.901,Z 479.527,A -85,B 0,C 180,E1 309.585,E2 309.585} C_VEL
LIN {X 0,Y 579.546,Z 470.468,A -85,B 0,C 180,E1 309.061,E2 309.061} C_VEL
LIN {X 0,Y 576.096,Z 459.907,A -85,B 0,C 180,E1 308.637,E2 308.637} C_VEL
LIN {X 0,Y 573.646,Z 447.926,A -85,B 0,C 180,E1 308.33,E2 308.33} C_VEL
LIN {X 0,Y 572.195,Z 434.184,A -85,B 0,C 180,E1 308.145,E2 308.145} C_VEL
LIN {X 0,Y 571.752,Z 419.101,A -85,B 0,C 180,E1 308.089,E2 308.089} C_VEL
LIN {X 0,Y 570.444,Z 420.274,A -85,B 0,C 180,E1 307.921,E2 307.921} C_VEL
LIN {X 0,Y 566.398,Z 430.589,A -85,B 0,C 180,E1 307.392,E2 307.392} C_VEL
LIN {X 0,Y 563.075,Z 436.308,A -85,B 0,C 180,E1 306.948,E2 306.948} C_VEL
LIN {X 0,Y 560.978,Z 438.035,A -85,B 0,C 180,E1 306.662,E2 306.662} C_VEL
LIN {X 0,Y 560.11,Z 437.943,A -85,B 0,C 180,E1 306.537,E2 306.537} C_VEL
LIN {X 0,Y 559.834,Z 455.36,A -85,B 0,C 180,E1 305.544,E2 305.544} C_VEL
LIN {X 0,Y 561.165,Z 465.397,A -85,B 0,C 180,E1 305.293,E2 305.293} C_VEL
LIN {X 0,Y 559.65,Z 681.144,A -85,B 0,C 180,E1 302.139,E2 302.139} C_VEL
LIN {X 0,Y 559.041,Z 761.898,A -85,B 0,C 180,E1 300.952,E2 300.952} C_VEL
LIN {X 0,Y 558.589,Z 784.038,A -85,B 0,C 180,E1 300.431,E2 300.431} C_VEL
LIN {X 0,Y 558.029,Z 806.457,A -85,B 0,C 180,E1 299.692,E2 299.692} C_VEL
LIN {X 0,Y 557.4,Z 827.558,A -85,B 0,C 180,E1 298.792,E2 298.792} C_VEL
LIN {X 0,Y 556.675,Z 847.765,A -85,B 0,C 180,E1 297.723,E2 297.723} C_VEL
LIN {X 0,Y 555.937,Z 867.641,A -85,B 0,C 180,E1 296.456,E2 296.456} C_VEL
LIN {X 0,Y 555.19,Z 886.467,A -85,B 0,C 180,E1 295.038,E2 295.038} C_VEL
LIN {X 0,Y 554.459,Z 905.27,A -85,B 0,C 180,E1 293.374,E2 293.374} C_VEL
LIN {X 0,Y 553.812,Z 922.336,A -85,B 0,C 180,E1 291.599,E2 291.599} C_VEL
LIN {X 0,Y 553.253,Z 938.113,A -85,B 0,C 180,E1 289.684,E2 289.684} C_VEL
LIN {X 0,Y 552.804,Z 952.175,A -85,B 0,C 180,E1 287.69,E2 287.69} C_VEL
LIN {X 0,Y 552.471,Z 964.524,A -85,B 0,C 180,E1 285.644,E2 285.644} C_VEL
LIN {X 0,Y 552.23,Z 975.404,A -85,B 0,C 180,E1 283.507,E2 283.507} C_VEL
LIN {X 0,Y 552.07,Z 984.311,A -85,B 0,C 180,E1 281.386,E2 281.386} C_VEL
LIN {X 0,Y 551.981,Z 992.176,A -85,B 0,C 180,E1 279.067,E2 279.067} C_VEL
LIN {X 0,Y 551.934,Z 997.921,A -85,B 0,C 180,E1 276.867,E2 276.867} C_VEL
LIN {X 0,Y 551.908,Z 1001.957,A -85,B 0,C 180,E1 274.676,E2 274.676} C_VEL
LIN {X 0,Y 551.904,Z 1004.556,A -85,B 0,C 180,E1 272.388,E2 272.388} C_VEL
LIN {X 0,Y 551.908,Z 1005.484,A -85,B 0,C 180,E1 270.104,E2 270.104} C_VEL
LIN {X 0,Y 551.913,Z 1004.762,A -85,B 0,C 180,E1 267.924,E2 267.924} C_VEL
LIN {X 0,Y 551.92,Z 1002.431,A -85,B 0,C 180,E1 265.637,E2 265.637} C_VEL
LIN {X 0,Y 551.937,Z 998.38,A -85,B 0,C 180,E1 263.343,E2 263.343} C_VEL
LIN {X 0,Y 551.97,Z 992.784,A -85,B 0,C 180,E1 261.143,E2 261.143} C_VEL
LIN {X 0,Y 552.058,Z 985.535,A -85,B 0,C 180,E1 258.932,E2 258.932} C_VEL
LIN {X 0,Y 552.215,Z 976.381,A -85,B 0,C 180,E1 256.706,E2 256.706} C_VEL
LIN {X 0,Y 552.447,Z 965.685,A -85,B 0,C 180,E1 254.571,E2 254.571} C_VEL
LIN {X 0,Y 552.79,Z 952.784,A -85,B 0,C 180,E1 252.403,E2 252.403} C_VEL
LIN {X 0,Y 553.217,Z 939.283,A -85,B 0,C 180,E1 250.467,E2 250.467} C_VEL
LIN {X 0,Y 553.777,Z 923.226,A -85,B 0,C 180,E1 248.499,E2 248.499} C_VEL
LIN {X 0,Y 554.436,Z 905.836,A -85,B 0,C 180,E1 246.682,E2 246.682} C_VEL
LIN {X 0,Y 555.144,Z 887.827,A -85,B 0,C 180,E1 245.074,E2 245.074} C_VEL
LIN {X 0,Y 555.907,Z 868.42,A -85,B 0,C 180,E1 243.599,E2 243.599} C_VEL
LIN {X 0,Y 556.652,Z 848.454,A -85,B 0,C 180,E1 242.316,E2 242.316} C_VEL
LIN {X 0,Y 557.358,Z 828.729,A -85,B 0,C 180,E1 241.264,E2 241.264} C_VEL
LIN {X 0,Y 557.991,Z 807.556,A -85,B 0,C 180,E1 240.35,E2 240.35} C_VEL
LIN {X 0,Y 558.575,Z 784.951,A -85,B 0,C 180,E1 239.595,E2 239.595} C_VEL
LIN {X 0,Y 559.019,Z 762.812,A -85,B 0,C 180,E1 239.066,E2 239.066} C_VEL
LIN {X 0,Y 559.433,Z 713.607,A -85,B 0,C 180,E1 238.328,E2 238.328} C_VEL
LIN {X 0,Y 560.965,Z 490.39,A -85,B 0,C 180,E1 235.076,E2 235.076} C_VEL
LIN {X 0,Y 560.975,Z 462.641,A -85,B 0,C 180,E1 234.651,E2 234.651} C_VEL
LIN {X 0,Y 559.723,Z 454.241,A -85,B 0,C 180,E1 234.416,E2 234.416} C_VEL
LIN {X 0,Y 560.229,Z 437.918,A -85,B 0,C 180,E1 233.441,E2 233.441} C_VEL
LIN {X 0,Y 561.722,Z 437.681,A -85,B 0,C 180,E1 233.236,E2 233.236} C_VEL
LIN {X 0,Y 564.351,Z 434.432,A -85,B 0,C 180,E1 232.88,E2 232.88} C_VEL
LIN {X 0,Y 568.068,Z 426.76,A -85,B 0,C 180,E1 232.388,E2 232.388} C_VEL
LIN {X 0,Y 570.671,Z 419.878,A -85,B 0,C 180,E1 232.05,E2 232.05} C_VEL
LIN {X 0,Y 571.763,Z 419.093,A -85,B 0,C 180,E1 231.91,E2 231.91} C_VEL
LIN {X 0,Y 572.308,Z 435.85,A -85,B 0,C 180,E1 231.84,E2 231.84} C_VEL
LIN {X 0,Y 573.875,Z 449.385,A -85,B 0,C 180,E1 231.642,E2 231.642} C_VEL
LIN {X 0,Y 576.444,Z 461.203,A -85,B 0,C 180,E1 231.32,E2 231.32} C_VEL
LIN {X 0,Y 580.093,Z 471.794,A -85,B 0,C 180,E1 230.872,E2 230.872} C_VEL
LIN {X 0,Y 584.615,Z 480.736,A -85,B 0,C 180,E1 230.33,E2 230.33} C_VEL
LIN {X 0,Y 589.06,Z 487.304,A -85,B 0,C 180,E1 229.771,E2 229.771} C_VEL
LIN {X 0,Y 591.07,Z 490.967,A -85,B 0,C 180,E1 229.274,E2 229.274} C_VEL
LIN {X 0,Y 591.736,Z 493.823,A -85,B 0,C 180,E1 228.681,E2 228.681} C_VEL
LIN {X 0,Y 590.955,Z 495.486,A -85,B 0,C 180,E1 228.063,E2 228.063} C_VEL
LIN {X 0,Y 588.897,Z 495.917,A -85,B 0,C 180,E1 227.465,E2 227.465} C_VEL
LIN {X 0,Y 585.867,Z 495.119,A -85,B 0,C 180,E1 226.923,E2 226.923} C_VEL
LIN {X 0,Y 580.883,Z 492.319,A -85,B 0,C 180,E1 226.297,E2 226.297} C_VEL
LIN {X 0,Y 574.942,Z 486.995,A -85,B 0,C 180,E1 225.48,E2 225.48} C_VEL
LIN {X 0,Y 570.346,Z 480.288,A -85,B 0,C 180,E1 224.666,E2 224.666} C_VEL
LIN {X 0,Y 567.039,Z 472.177,A -85,B 0,C 180,E1 223.848,E2 223.848} C_VEL
LIN {X 0,Y 564.916,Z 461.843,A -85,B 0,C 180,E1 222.954,E2 222.954} C_VEL
LIN {X 0,Y 564.002,Z 448.302,A -85,B 0,C 180,E1 221.939,E2 221.939} C_VEL
LIN {X 0,Y 565.622,Z 396.546,A -85,B 0,C 180,E1 218.455,E2 218.455} C_VEL
LIN {X 0,Y 565.932,Z 387.444,A -85,B 0,C 180,E1 217.811,E2 217.811} C_VEL
LIN {X 0,Y 559.933,Z 376.207,A -85,B 0,C 180,E1 216.232,E2 216.232} C_VEL
LIN {X 0,Y 556.913,Z 370.994,A -85,B 0,C 180,E1 215.443,E2 215.443} C_VEL
LIN {X 0,Y 554.374,Z 366.395,A -85,B 0,C 180,E1 214.745,E2 214.745} C_VEL
LIN {X 0,Y 552.571,Z 363.085,A -85,B 0,C 180,E1 214.245,E2 214.245} C_VEL
LIN {X 0,Y 552.339,Z 361.927,A -85,B 0,C 180,E1 214.111,E2 214.111} C_VEL
LIN {X 0,Y 552.335,Z 361.937,A -85,B 0,C 180,E1 210.817,E2 210.817} C_VEL
LIN {X 0,Y 552.314,Z 361.937,A -85,B 0,C 180,E1 207.492,E2 207.492} C_VEL
LIN {X 0,Y 552.337,Z 361.934,A -85,B 0,C 180,E1 204.167,E2 204.167} C_VEL
LIN {X 0,Y 552.298,Z 361.937,A -85,B 0,C 180,E1 200.783,E2 200.783} C_VEL
LIN {X 0,Y 552.33,Z 361.932,A -85,B 0,C 180,E1 197.379,E2 197.379} C_VEL
LIN {X 0,Y 552.309,Z 361.935,A -85,B 0,C 180,E1 194.146,E2 194.146} C_VEL
LIN {X 0,Y 552.301,Z 361.937,A -85,B 0,C 180,E1 190.641,E2 190.641} C_VEL
LIN {X 0,Y 552.338,Z 361.932,A -85,B 0,C 180,E1 187.384,E2 187.384} C_VEL
LIN {X 0,Y 552.293,Z 361.938,A -85,B 0,C 180,E1 184.041,E2 184.041} C_VEL
LIN {X 0,Y 552.334,Z 361.935,A -85,B 0,C 180,E1 180.622,E2 180.622} C_VEL
LIN {X 0,Y 552.299,Z 361.939,A -85,B 0,C 180,E1 177.406,E2 177.406} C_VEL
LIN {X 0,Y 552.324,Z 361.935,A -85,B 0,C 180,E1 174.077,E2 174.077} C_VEL
LIN {X 0,Y 552.339,Z 361.936,A -85,B 0,C 180,E1 170.728,E2 170.728} C_VEL
LIN {X 0,Y 552.329,Z 361.938,A -85,B 0,C 180,E1 167.347,E2 167.347} C_VEL
LIN {X 0,Y 552.339,Z 361.936,A -85,B 0,C 180,E1 163.993,E2 163.993} C_VEL
LIN {X 0,Y 552.344,Z 361.935,A -85,B 0,C 180,E1 160.544,E2 160.544} C_VEL
LIN {X 0,Y 552.322,Z 361.935,A -85,B 0,C 180,E1 157.136,E2 157.136} C_VEL
LIN {X 0,Y 552.31,Z 361.935,A -85,B 0,C 180,E1 153.786,E2 153.786} C_VEL
LIN {X 0,Y 552.328,Z 361.935,A -85,B 0,C 180,E1 152.719,E2 152.719} C_VEL
LIN {X 0,Y 551.384,Z 362.053,A -85,B 0,C 180,E1 151.92,E2 151.92} C_VEL
LIN {X 0,Y 544.851,Z 362.868,A -85,B 0,C 180,E1 149.618,E2 149.618} C_VEL
LIN {X 0,Y 544.382,Z 362.922,A -85,B 0,C 180,E1 149.092,E2 149.092} C_VEL
LIN {X 0,Y 544.387,Z 362.921,A -85,B 0,C 180,E1 145.677,E2 145.677} C_VEL
LIN {X 0,Y 544.382,Z 362.919,A -85,B 0,C 180,E1 142.336,E2 142.336} C_VEL
LIN {X 0,Y 544.35,Z 362.923,A -85,B 0,C 180,E1 138.858,E2 138.858} C_VEL
LIN {X 0,Y 544.402,Z 362.922,A -85,B 0,C 180,E1 135.593,E2 135.593} C_VEL
LIN {X 0,Y 544.351,Z 362.923,A -85,B 0,C 180,E1 132.242,E2 132.242} C_VEL
LIN {X 0,Y 544.386,Z 362.918,A -85,B 0,C 180,E1 128.778,E2 128.778} C_VEL
LIN {X 0,Y 544.378,Z 362.927,A -85,B 0,C 180,E1 125.478,E2 125.478} C_VEL
LIN {X 0,Y 544.429,Z 363.119,A -85,B 0,C 180,E1 123.319,E2 123.319} C_VEL
LIN {X 0,Y 550.127,Z 379.154,A -85,B 0,C 180,E1 121.764,E2 121.764} C_VEL
LIN {X 0,Y 549.189,Z 424.152,A -85,B 0,C 180,E1 118.489,E2 118.489} C_VEL
LIN {X 0,Y 548.127,Z 466.985,A -85,B 0,C 180,E1 115.383,E2 115.383} C_VEL
LIN {X 0,Y 548.02,Z 474.216,A -85,B 0,C 180,E1 114.874,E2 114.874} C_VEL
LIN {X 0,Y 549.128,Z 483.4,A -85,B 0,C 180,E1 114.687,E2 114.687} C_VEL
LIN {X 0,Y 547.995,Z 682.351,A -85,B 0,C 180,E1 111.926,E2 111.926} C_VEL
LIN {X 0,Y 547.703,Z 701.063,A -85,B 0,C 180,E1 111.48,E2 111.48} C_VEL
LIN {X 0,Y 547.325,Z 718.783,A -85,B 0,C 180,E1 110.868,E2 110.868} C_VEL
LIN {X 0,Y 546.845,Z 736.704,A -85,B 0,C 180,E1 110.049,E2 110.049} C_VEL
LIN {X 0,Y 546.342,Z 754.052,A -85,B 0,C 180,E1 109.039,E2 109.039} C_VEL
LIN {X 0,Y 545.855,Z 770.292,A -85,B 0,C 180,E1 107.867,E2 107.867} C_VEL
LIN {X 0,Y 545.358,Z 785.74,A -85,B 0,C 180,E1 106.509,E2 106.509} C_VEL
LIN {X 0,Y 544.922,Z 800.01,A -85,B 0,C 180,E1 104.994,E2 104.994} C_VEL
LIN {X 0,Y 544.572,Z 812.646,A -85,B 0,C 180,E1 103.376,E2 103.376} C_VEL
LIN {X 0,Y 544.304,Z 823.739,A -85,B 0,C 180,E1 101.657,E2 101.657} C_VEL
LIN {X 0,Y 544.121,Z 833.306,A -85,B 0,C 180,E1 99.839,E2 99.839} C_VEL
LIN {X 0,Y 544.001,Z 840.914,A -85,B 0,C 180,E1 98.029,E2 98.029} C_VEL
LIN {X 0,Y 543.947,Z 847.087,A -85,B 0,C 180,E1 96.12,E2 96.12} C_VEL
LIN {X 0,Y 543.923,Z 851.491,A -85,B 0,C 180,E1 94.216,E2 94.216} C_VEL
LIN {X 0,Y 543.915,Z 854.354,A -85,B 0,C 180,E1 92.212,E2 92.212} C_VEL
LIN {X 0,Y 543.912,Z 855.452,A -85,B 0,C 180,E1 90.21,E2 90.21} C_VEL
LIN {X 0,Y 543.913,Z 854.809,A -85,B 0,C 180,E1 88.209,E2 88.209} C_VEL
LIN {X 0,Y 543.917,Z 852.414,A -85,B 0,C 180,E1 86.205,E2 86.205} C_VEL
LIN {X 0,Y 543.932,Z 848.454,A -85,B 0,C 180,E1 84.303,E2 84.303} C_VEL
LIN {X 0,Y 543.985,Z 842.77,A -85,B 0,C 180,E1 82.395,E2 82.395} C_VEL
LIN {X 0,Y 544.084,Z 835.211,A -85,B 0,C 180,E1 80.48,E2 80.48} C_VEL
LIN {X 0,Y 544.255,Z 826.119,A -85,B 0,C 180,E1 78.663,E2 78.663} C_VEL
LIN {X 0,Y 544.503,Z 815.546,A -85,B 0,C 180,E1 76.946,E2 76.946} C_VEL
LIN {X 0,Y 544.839,Z 802.977,A -85,B 0,C 180,E1 75.268,E2 75.268} C_VEL
LIN {X 0,Y 545.248,Z 789.361,A -85,B 0,C 180,E1 73.76,E2 73.76} C_VEL
LIN {X 0,Y 545.713,Z 774.637,A -85,B 0,C 180,E1 72.403,E2 72.403} C_VEL
LIN {X 0,Y 546.229,Z 758.131,A -85,B 0,C 180,E1 71.149,E2 71.149} C_VEL
LIN {X 0,Y 546.703,Z 741.36,A -85,B 0,C 180,E1 70.112,E2 70.112} C_VEL
LIN {X 0,Y 547.207,Z 723.525,A -85,B 0,C 180,E1 69.238,E2 69.238} C_VEL
LIN {X 0,Y 547.626,Z 704.88,A -85,B 0,C 180,E1 68.545,E2 68.545} C_VEL
LIN {X 0,Y 547.951,Z 685.726,A -85,B 0,C 180,E1 68.047,E2 68.047} C_VEL
LIN {X 0,Y 548.162,Z 657.746,A -85,B 0,C 180,E1 67.621,E2 67.621} C_VEL
LIN {X 0,Y 548.962,Z 480.408,A -85,B 0,C 180,E1 65.172,E2 65.172} C_VEL
LIN {X 0,Y 547.947,Z 473.464,A -85,B 0,C 180,E1 65.008,E2 65.008} C_VEL
LIN {X 0,Y 549.057,Z 429.565,A -85,B 0,C 180,E1 61.811,E2 61.811} C_VEL
LIN {X 0,Y 550.005,Z 386.408,A -85,B 0,C 180,E1 58.673,E2 58.673} C_VEL
LIN {X 0,Y 549.994,Z 378.665,A -85,B 0,C 180,E1 58.101,E2 58.101} C_VEL
LIN {X 0,Y 544.367,Z 362.927,A -85,B 0,C 180,E1 56.563,E2 56.563} C_VEL
LIN {X 0,Y 544.371,Z 362.929,A -85,B 0,C 180,E1 53.384,E2 53.384} C_VEL
LIN {X 0,Y 544.345,Z 362.923,A -85,B 0,C 180,E1 49.992,E2 49.992} C_VEL
LIN {X 0,Y 544.405,Z 362.92,A -85,B 0,C 180,E1 46.76,E2 46.76} C_VEL
LIN {X 0,Y 544.342,Z 362.927,A -85,B 0,C 180,E1 43.485,E2 43.485} C_VEL
LIN {X 0,Y 544.378,Z 362.923,A -85,B 0,C 180,E1 40.142,E2 40.142} C_VEL
LIN {X 0,Y 544.361,Z 362.929,A -85,B 0,C 180,E1 36.915,E2 36.915} C_VEL
LIN {X 0,Y 544.359,Z 362.942,A -85,B 0,C 180,E1 35.772,E2 35.772} C_VEL
LIN {X 0,Y 551.485,Z 381.845,A -85,B 0,C 180,E1 33.64,E2 33.64} C_VEL
LIN {X 0,Y 550.46,Z 418.916,A -85,B 0,C 180,E1 30.691,E2 30.691} C_VEL
LIN {X 0,Y 549.116,Z 462.672,A -85,B 0,C 180,E1 27.255,E2 27.255} C_VEL
LIN {X 0,Y 547.924,Z 508.06,A -85,B 0,C 180,E1 23.784,E2 23.784} C_VEL
LIN {X 0,Y 546.63,Z 555.21,A -85,B 0,C 180,E1 20.169,E2 20.169} C_VEL
LIN {X 0,Y 545.927,Z 589.13,A -85,B 0,C 180,E1 17.647,E2 17.647} C_VEL
LIN {X 0,Y 546.544,Z 597.733,A -85,B 0,C 180,E1 17.506,E2 17.506} C_VEL
LIN {X 0,Y 545.99,Z 730.5,A -85,B 0,C 180,E1 15.709,E2 15.709} C_VEL
LIN {X 0,Y 545.83,Z 746.157,A -85,B 0,C 180,E1 15.335,E2 15.335} C_VEL
LIN {X 0,Y 545.582,Z 761.523,A -85,B 0,C 180,E1 14.758,E2 14.758} C_VEL
LIN {X 0,Y 545.339,Z 773.519,A -85,B 0,C 180,E1 14.168,E2 14.168} C_VEL
LIN {X 0,Y 545.084,Z 785.773,A -85,B 0,C 180,E1 13.418,E2 13.418} C_VEL
LIN {X 0,Y 544.789,Z 799.745,A -85,B 0,C 180,E1 12.346,E2 12.346} C_VEL
LIN {X 0,Y 544.523,Z 811.315,A -85,B 0,C 180,E1 11.224,E2 11.224} C_VEL
LIN {X 0,Y 544.321,Z 821.119,A -85,B 0,C 180,E1 10.075,E2 10.075} C_VEL
LIN {X 0,Y 544.135,Z 831.536,A -85,B 0,C 180,E1 8.56,E2 8.56} C_VEL
LIN {X 0,Y 544.026,Z 838.961,A -85,B 0,C 180,E1 7.18,E2 7.18} C_VEL
LIN {X 0,Y 543.964,Z 844.858,A -85,B 0,C 180,E1 5.803,E2 5.803} C_VEL
LIN {X 0,Y 543.928,Z 850.226,A -85,B 0,C 180,E1 4.111,E2 4.111} C_VEL
LIN {X 0,Y 543.917,Z 853.427,A -85,B 0,C 180,E1 2.529,E2 2.529} C_VEL
LIN {X 0,Y 543.916,Z 855.071,A -85,B 0,C 180,E1 1.054,E2 1.054} C_VEL
LIN {X 0,Y 543.915,Z 855.392,A -85,B 0,C 180,E1 -0.632,E2 -0.632} C_VEL
LIN {X 0,Y 543.915,Z 853.879,A -85,B 0,C 180,E1 -2.317,E2 -2.317} C_VEL
LIN {X 0,Y 543.922,Z 851.162,A -85,B 0,C 180,E1 -3.794,E2 -3.794} C_VEL
LIN {X 0,Y 543.95,Z 846.734,A -85,B 0,C 180,E1 -5.379,E2 -5.379} C_VEL
LIN {X 0,Y 544.012,Z 840.131,A -85,B 0,C 180,E1 -7.025,E2 -7.025} C_VEL
LIN {X 0,Y 544.104,Z 833.277,A -85,B 0,C 180,E1 -8.347,E2 -8.347} C_VEL
LIN {X 0,Y 544.262,Z 824.415,A -85,B 0,C 180,E1 -9.73,E2 -9.73} C_VEL
LIN {X 0,Y 544.484,Z 813.152,A -85,B 0,C 180,E1 -11.117,E2 -11.117} C_VEL
LIN {X 0,Y 544.719,Z 802.474,A -85,B 0,C 180,E1 -12.186,E2 -12.186} C_VEL
LIN {X 0,Y 544.996,Z 790.164,A -85,B 0,C 180,E1 -13.203,E2 -13.203} C_VEL
LIN {X 0,Y 545.293,Z 776.121,A -85,B 0,C 180,E1 -14.115,E2 -14.115} C_VEL
LIN {X 0,Y 545.543,Z 763.518,A -85,B 0,C 180,E1 -14.759,E2 -14.759} C_VEL
LIN {X 0,Y 545.747,Z 750.678,A -85,B 0,C 180,E1 -15.269,E2 -15.269} C_VEL
LIN {X 0,Y 545.966,Z 734.889,A -85,B 0,C 180,E1 -15.719,E2 -15.719} C_VEL
LIN {X 0,Y 546.118,Z 710.252,A -85,B 0,C 180,E1 -16.095,E2 -16.095} C_VEL
LIN {X 0,Y 546.424,Z 592.884,A -85,B 0,C 180,E1 -17.691,E2 -17.691} C_VEL
LIN {X 0,Y 546.153,Z 590.268,A -85,B 0,C 180,E1 -17.747,E2 -17.747} C_VEL
LIN {X 0,Y 547.797,Z 553.699,A -85,B 0,C 180,E1 -20.682,E2 -20.682} C_VEL
LIN {X 0,Y 550.34,Z 510.902,A -85,B 0,C 180,E1 -24.211,E2 -24.211} C_VEL
LIN {X 0,Y 553.383,Z 472.139,A -85,B 0,C 180,E1 -27.551,E2 -27.551} C_VEL
LIN {X 0,Y 557.38,Z 437.589,A -85,B 0,C 180,E1 -30.687,E2 -30.687} C_VEL
LIN {X 0,Y 561.981,Z 410.257,A -85,B 0,C 180,E1 -33.35,E2 -33.35} C_VEL
LIN {X 0,Y 563.476,Z 402.769,A -85,B 0,C 180,E1 -34.167,E2 -34.167} C_VEL
LIN {X 0,Y 564.367,Z 398.115,A -85,B 0,C 180,E1 -34.748,E2 -34.748} C_VEL
LIN {X 0,Y 563.336,Z 394.943,A -85,B 0,C 180,E1 -35.794,E2 -35.794} C_VEL
LIN {X 0,Y 563.033,Z 392.813,A -85,B 0,C 180,E1 -37.014,E2 -37.014} C_VEL
LIN {X 0,Y 563.316,Z 392.475,A -85,B 0,C 180,E1 -37.503,E2 -37.503} C_VEL
LIN {X 0,Y 563.158,Z 393.518,A -85,B 0,C 180,E1 -37.93,E2 -37.93} C_VEL
LIN {X 0,Y 559.018,Z 404.798,A -85,B 0,C 180,E1 -38.918,E2 -38.918} C_VEL
LIN {X 0,Y 555.773,Z 419.415,A -85,B 0,C 180,E1 -40.049,E2 -40.049} C_VEL
LIN {X 0,Y 553.642,Z 438.264,A -85,B 0,C 180,E1 -41.375,E2 -41.375} C_VEL
LIN {X 0,Y 553.74,Z 453.917,A -85,B 0,C 180,E1 -42.478,E2 -42.478} C_VEL
LIN {X 0,Y 555.768,Z 467.375,A -85,B 0,C 180,E1 -43.483,E2 -43.483} C_VEL
LIN {X 0,Y 559.292,Z 478.047,A -85,B 0,C 180,E1 -44.346,E2 -44.346} C_VEL
LIN {X 0,Y 564.276,Z 486.903,A -85,B 0,C 180,E1 -45.135,E2 -45.135} C_VEL
LIN {X 0,Y 570.857,Z 494.452,A -85,B 0,C 180,E1 -45.899,E2 -45.899} C_VEL
LIN {X 0,Y 578.894,Z 500.492,A -85,B 0,C 180,E1 -46.647,E2 -46.647} C_VEL
LIN {X 0,Y 582.839,Z 502.426,A -85,B 0,C 180,E1 -47.097,E2 -47.097} C_VEL
LIN {X 0,Y 586.176,Z 503.251,A -85,B 0,C 180,E1 -47.641,E2 -47.641} C_VEL
LIN {X 0,Y 588.457,Z 502.871,A -85,B 0,C 180,E1 -48.237,E2 -48.237} C_VEL
LIN {X 0,Y 589.452,Z 501.295,A -85,B 0,C 180,E1 -48.862,E2 -48.862} C_VEL
LIN {X 0,Y 589.009,Z 498.685,A -85,B 0,C 180,E1 -49.446,E2 -49.446} C_VEL
LIN {X 0,Y 587.172,Z 495.239,A -85,B 0,C 180,E1 -49.965,E2 -49.965} C_VEL
LIN {X 0,Y 583.424,Z 490.05,A -85,B 0,C 180,E1 -50.472,E2 -50.472} C_VEL
LIN {X 0,Y 578.366,Z 481.575,A -85,B 0,C 180,E1 -51.083,E2 -51.083} C_VEL
LIN {X 0,Y 574.073,Z 471.41,A -85,B 0,C 180,E1 -51.617,E2 -51.617} C_VEL
LIN {X 0,Y 570.79,Z 460.027,A -85,B 0,C 180,E1 -52.035,E2 -52.035} C_VEL
LIN {X 0,Y 568.471,Z 447.099,A -85,B 0,C 180,E1 -52.335,E2 -52.335} C_VEL
LIN {X 0,Y 567.613,Z 440.358,A -85,B 0,C 180,E1 -52.447,E2 -52.447} C_VEL
LIN {X 0,Y 564.279,Z 444.51,A -85,B 0,C 180,E1 -52.89,E2 -52.89} C_VEL
LIN {X 0,Y 563.112,Z 445.656,A -85,B 0,C 180,E1 -53.047,E2 -53.047} C_VEL
LIN {X 0,Y 559.044,Z 456.445,A -85,B 0,C 180,E1 -53.605,E2 -53.605} C_VEL
LIN {X 0,Y 556.312,Z 463.924,A -85,B 0,C 180,E1 -53.989,E2 -53.989} C_VEL
LIN {X 0,Y 555.066,Z 465.285,A -85,B 0,C 180,E1 -54.166,E2 -54.166} C_VEL
LIN {X 0,Y 554.634,Z 465.574,A -85,B 0,C 180,E1 -54.231,E2 -54.231} C_VEL
LIN {X 0,Y 552.874,Z 681.297,A -85,B 0,C 180,E1 -57.421,E2 -57.421} C_VEL
LIN {X 0,Y 552.174,Z 761.885,A -85,B 0,C 180,E1 -58.62,E2 -58.62} C_VEL
LIN {X 0,Y 551.654,Z 784.006,A -85,B 0,C 180,E1 -59.144,E2 -59.144} C_VEL
LIN {X 0,Y 551.029,Z 806.316,A -85,B 0,C 180,E1 -59.886,E2 -59.886} C_VEL
LIN {X 0,Y 550.289,Z 827.553,A -85,B 0,C 180,E1 -60.8,E2 -60.8} C_VEL
LIN {X 0,Y 549.466,Z 847.772,A -85,B 0,C 180,E1 -61.881,E2 -61.881} C_VEL
LIN {X 0,Y 548.594,Z 867.974,A -85,B 0,C 180,E1 -63.186,E2 -63.186} C_VEL
LIN {X 0,Y 547.719,Z 886.949,A -85,B 0,C 180,E1 -64.637,E2 -64.637} C_VEL
LIN {X 0,Y 546.901,Z 905.27,A -85,B 0,C 180,E1 -66.283,E2 -66.283} C_VEL
LIN {X 0,Y 546.122,Z 923.034,A -85,B 0,C 180,E1 -68.16,E2 -68.16} C_VEL
LIN {X 0,Y 545.451,Z 939.279,A -85,B 0,C 180,E1 -70.176,E2 -70.176} C_VEL
LIN {X 0,Y 544.921,Z 953.593,A -85,B 0,C 180,E1 -72.266,E2 -72.266} C_VEL
LIN {X 0,Y 544.527,Z 966.264,A -85,B 0,C 180,E1 -74.449,E2 -74.449} C_VEL
LIN {X 0,Y 544.259,Z 976.85,A -85,B 0,C 180,E1 -76.616,E2 -76.616} C_VEL
LIN {X 0,Y 544.079,Z 985.924,A -85,B 0,C 180,E1 -78.874,E2 -78.874} C_VEL
LIN {X 0,Y 543.98,Z 993.09,A -85,B 0,C 180,E1 -81.118,E2 -81.118} C_VEL
LIN {X 0,Y 543.936,Z 998.798,A -85,B 0,C 180,E1 -83.456,E2 -83.456} C_VEL
LIN {X 0,Y 543.919,Z 1002.736,A -85,B 0,C 180,E1 -85.783,E2 -85.783} C_VEL
LIN {X 0,Y 543.907,Z 1004.897,A -85,B 0,C 180,E1 -88.103,E2 -88.103} C_VEL
LIN {X 0,Y 543.893,Z 1005.417,A -85,B 0,C 180,E1 -90.526,E2 -90.526} C_VEL
LIN {X 0,Y 543.892,Z 1004.332,A -85,B 0,C 180,E1 -92.739,E2 -92.739} C_VEL
LIN {X 0,Y 543.899,Z 1001.643,A -85,B 0,C 180,E1 -94.956,E2 -94.956} C_VEL
LIN {X 0,Y 543.924,Z 997.188,A -85,B 0,C 180,E1 -97.287,E2 -97.287} C_VEL
LIN {X 0,Y 543.989,Z 991.254,A -85,B 0,C 180,E1 -99.521,E2 -99.521} C_VEL
LIN {X 0,Y 544.108,Z 983.502,A -85,B 0,C 180,E1 -101.769,E2 -101.769} C_VEL
LIN {X 0,Y 544.313,Z 973.871,A -85,B 0,C 180,E1 -104.032,E2 -104.032} C_VEL
LIN {X 0,Y 544.626,Z 962.602,A -85,B 0,C 180,E1 -106.229,E2 -106.229} C_VEL
LIN {X 0,Y 545.067,Z 949.345,A -85,B 0,C 180,E1 -108.392,E2 -108.392} C_VEL
LIN {X 0,Y 545.605,Z 935.045,A -85,B 0,C 180,E1 -110.376,E2 -110.376} C_VEL
LIN {X 0,Y 546.273,Z 919.222,A -85,B 0,C 180,E1 -112.264,E2 -112.264} C_VEL
LIN {X 0,Y 547.06,Z 901.737,A -85,B 0,C 180,E1 -114.052,E2 -114.052} C_VEL
LIN {X 0,Y 547.895,Z 883.543,A -85,B 0,C 180,E1 -115.644,E2 -115.644} C_VEL
LIN {X 0,Y 548.769,Z 863.948,A -85,B 0,C 180,E1 -117.097,E2 -117.097} C_VEL
LIN {X 0,Y 549.626,Z 843.804,A -85,B 0,C 180,E1 -118.346,E2 -118.346} C_VEL
LIN {X 0,Y 550.458,Z 822.673,A -85,B 0,C 180,E1 -119.428,E2 -119.428} C_VEL
LIN {X 0,Y 551.194,Z 801.512,A -85,B 0,C 180,E1 -120.294,E2 -120.294} C_VEL
LIN {X 0,Y 551.784,Z 779.494,A -85,B 0,C 180,E1 -120.98,E2 -120.98} C_VEL
LIN {X 0,Y 552.233,Z 757.571,A -85,B 0,C 180,E1 -121.457,E2 -121.457} C_VEL
LIN {X 0,Y 554.076,Z 531.938,A -85,B 0,C 180,E1 -124.778,E2 -124.778} C_VEL
LIN {X 0,Y 554.77,Z 465.341,A -85,B 0,C 180,E1 -125.792,E2 -125.792} C_VEL
LIN {X 0,Y 556.162,Z 464.183,A -85,B 0,C 180,E1 -125.99,E2 -125.99} C_VEL
LIN {X 0,Y 558.004,Z 459.471,A -85,B 0,C 180,E1 -126.25,E2 -126.25} C_VEL
LIN {X 0,Y 559.282,Z 455.911,A -85,B 0,C 180,E1 -126.428,E2 -126.428} C_VEL
LIN {X 0,Y 563.371,Z 445.196,A -85,B 0,C 180,E1 -126.988,E2 -126.988} C_VEL
LIN {X 0,Y 566.47,Z 442.054,A -85,B 0,C 180,E1 -127.402,E2 -127.402} C_VEL
LIN {X 0,Y 567.725,Z 440.387,A -85,B 0,C 180,E1 -127.567,E2 -127.567} C_VEL
LIN {X 0,Y 569.577,Z 454.153,A -85,B 0,C 180,E1 -127.809,E2 -127.809} C_VEL
LIN {X 0,Y 572.405,Z 466.217,A -85,B 0,C 180,E1 -128.172,E2 -128.172} C_VEL
LIN {X 0,Y 576.171,Z 476.829,A -85,B 0,C 180,E1 -128.646,E2 -128.646} C_VEL
LIN {X 0,Y 580.962,Z 486.299,A -85,B 0,C 180,E1 -129.233,E2 -129.233} C_VEL
LIN {X 0,Y 586.415,Z 494.124,A -85,B 0,C 180,E1 -129.905,E2 -129.905} C_VEL
LIN {X 0,Y 588.686,Z 497.924,A -85,B 0,C 180,E1 -130.42,E2 -130.42} C_VEL
LIN {X 0,Y 589.474,Z 500.758,A -85,B 0,C 180,E1 -130.992,E2 -130.992} C_VEL
LIN {X 0,Y 588.857,Z 502.57,A -85,B 0,C 180,E1 -131.598,E2 -131.598} C_VEL
LIN {X 0,Y 586.976,Z 503.265,A -85,B 0,C 180,E1 -132.185,E2 -132.185} C_VEL
LIN {X 0,Y 584.002,Z 502.812,A -85,B 0,C 180,E1 -132.737,E2 -132.737} C_VEL
LIN {X 0,Y 579.624,Z 500.91,A -85,B 0,C 180,E1 -133.285,E2 -133.285} C_VEL
LIN {X 0,Y 572.541,Z 495.9,A -85,B 0,C 180,E1 -134.17,E2 -134.17} C_VEL
LIN {X 0,Y 567.148,Z 489.765,A -85,B 0,C 180,E1 -135.013,E2 -135.013} C_VEL
LIN {X 0,Y 562.721,Z 481.671,A -85,B 0,C 180,E1 -135.923,E2 -135.923} C_VEL
LIN {X 0,Y 559.787,Z 472.105,A -85,B 0,C 180,E1 -136.836,E2 -136.836} C_VEL
LIN {X 0,Y 558.026,Z 458.817,A -85,B 0,C 180,E1 -137.924,E2 -137.924} C_VEL
LIN {X 0,Y 557.974,Z 441.444,A -85,B 0,C 180,E1 -139.152,E2 -139.152} C_VEL
LIN {X 0,Y 559.69,Z 400.257,A -85,B 0,C 180,E1 -141.952,E2 -141.952} C_VEL
LIN {X 0,Y 560.004,Z 391.791,A -85,B 0,C 180,E1 -142.559,E2 -142.559} C_VEL
LIN {X 0,Y 551.951,Z 377.115,A -85,B 0,C 180,E1 -144.7,E2 -144.7} C_VEL
LIN {X 0,Y 548.96,Z 371.981,A -85,B 0,C 180,E1 -145.498,E2 -145.498} C_VEL
LIN {X 0,Y 546.9,Z 367.813,A -85,B 0,C 180,E1 -146.11,E2 -146.11} C_VEL
LIN {X 0,Y 544.94,Z 365.069,A -85,B 0,C 180,E1 -146.603,E2 -146.603} C_VEL
LIN {X 0,Y 544.364,Z 362.918,A -85,B 0,C 180,E1 -146.883,E2 -146.883} C_VEL
LIN {X 0,Y 544.403,Z 362.923,A -85,B 0,C 180,E1 -150.31,E2 -150.31} C_VEL
LIN {X 0,Y 544.384,Z 362.927,A -85,B 0,C 180,E1 -153.675,E2 -153.675} C_VEL
LIN {X 0,Y 544.405,Z 362.923,A -85,B 0,C 180,E1 -157.086,E2 -157.086} C_VEL
LIN {X 0,Y 544.387,Z 362.924,A -85,B 0,C 180,E1 -160.472,E2 -160.472} C_VEL
LIN {X 0,Y 544.397,Z 362.922,A -85,B 0,C 180,E1 -163.854,E2 -163.854} C_VEL
LIN {X 0,Y 544.363,Z 362.927,A -85,B 0,C 180,E1 -167.267,E2 -167.267} C_VEL
LIN {X 0,Y 544.404,Z 362.922,A -85,B 0,C 180,E1 -170.593,E2 -170.593} C_VEL
LIN {X 0,Y 544.363,Z 362.925,A -85,B 0,C 180,E1 -173.885,E2 -173.885} C_VEL
LIN {X 0,Y 544.376,Z 362.925,A -85,B 0,C 180,E1 -177.368,E2 -177.368} C_VEL
LIN {X 0,Y 544.38,Z 362.923,A -85,B 0,C 180,E1 -180.632,E2 -180.632} C_VEL
LIN {X 0,Y 544.359,Z 362.928,A -85,B 0,C 180,E1 -184.108,E2 -184.108} C_VEL
LIN {X 0,Y 544.402,Z 362.923,A -85,B 0,C 180,E1 -187.493,E2 -187.493} C_VEL
LIN {X 0,Y 544.366,Z 362.926,A -85,B 0,C 180,E1 -190.798,E2 -190.798} C_VEL
LIN {X 0,Y 544.392,Z 362.925,A -85,B 0,C 180,E1 -194.139,E2 -194.139} C_VEL
LIN {X 0,Y 544.395,Z 362.926,A -85,B 0,C 180,E1 -197.531,E2 -197.531} C_VEL
LIN {X 0,Y 544.401,Z 362.924,A -85,B 0,C 180,E1 -200.874,E2 -200.874} C_VEL
LIN {X 0,Y 544.399,Z 362.924,A -85,B 0,C 180,E1 -204.178,E2 -204.178} C_VEL
LIN {X 0,Y 544.406,Z 362.921,A -85,B 0,C 180,E1 -207.57,E2 -207.57} C_VEL
LIN {X 0,Y 544.382,Z 362.922,A -85,B 0,C 180,E1 -210.908,E2 -210.908} C_VEL
LIN {X 0,Y 543.364,Z 363.047,A -85,B 0,C 180,E1 -211.719,E2 -211.719} C_VEL
LIN {X 0,Y 536.974,Z 363.848,A -85,B 0,C 180,E1 -213.995,E2 -213.995} C_VEL
LIN {X 0,Y 536.433,Z 363.91,A -85,B 0,C 180,E1 -214.588,E2 -214.588} C_VEL
LIN {X 0,Y 536.444,Z 363.907,A -85,B 0,C 180,E1 -217.822,E2 -217.822} C_VEL
LIN {X 0,Y 536.413,Z 363.912,A -85,B 0,C 180,E1 -221.308,E2 -221.308} C_VEL
LIN {X 0,Y 536.461,Z 363.912,A -85,B 0,C 180,E1 -224.757,E2 -224.757} C_VEL
LIN {X 0,Y 536.424,Z 363.911,A -85,B 0,C 180,E1 -228.049,E2 -228.049} C_VEL
LIN {X 0,Y 536.45,Z 363.905,A -85,B 0,C 180,E1 -231.363,E2 -231.363} C_VEL
LIN {X 0,Y 536.453,Z 363.916,A -85,B 0,C 180,E1 -234.722,E2 -234.722} C_VEL
LIN {X 0,Y 536.444,Z 364.062,A -85,B 0,C 180,E1 -236.196,E2 -236.196} C_VEL
LIN {X 0,Y 543.011,Z 382.021,A -85,B 0,C 180,E1 -237.974,E2 -237.974} C_VEL
LIN {X 0,Y 541.912,Z 427.704,A -85,B 0,C 180,E1 -241.334,E2 -241.334} C_VEL
LIN {X 0,Y 540.768,Z 473.477,A -85,B 0,C 180,E1 -244.657,E2 -244.657} C_VEL
LIN {X 0,Y 540.883,Z 475.755,A -85,B 0,C 180,E1 -244.78,E2 -244.78} C_VEL
LIN {X 0,Y 541.915,Z 484.53,A -85,B 0,C 180,E1 -244.961,E2 -244.961} C_VEL
LIN {X 0,Y 540.577,Z 682.448,A -85,B 0,C 180,E1 -247.757,E2 -247.757} C_VEL
LIN {X 0,Y 540.238,Z 701.267,A -85,B 0,C 180,E1 -248.214,E2 -248.214} C_VEL
LIN {X 0,Y 539.802,Z 719.458,A -85,B 0,C 180,E1 -248.854,E2 -248.854} C_VEL
LIN {X 0,Y 539.247,Z 737.802,A -85,B 0,C 180,E1 -249.713,E2 -249.713} C_VEL
LIN {X 0,Y 538.688,Z 754.486,A -85,B 0,C 180,E1 -250.708,E2 -250.708} C_VEL
LIN {X 0,Y 538.121,Z 770.964,A -85,B 0,C 180,E1 -251.923,E2 -251.923} C_VEL
LIN {X 0,Y 537.581,Z 785.749,A -85,B 0,C 180,E1 -253.245,E2 -253.245} C_VEL
LIN {X 0,Y 537.114,Z 799.101,A -85,B 0,C 180,E1 -254.673,E2 -254.673} C_VEL
LIN {X 0,Y 536.7,Z 811.889,A -85,B 0,C 180,E1 -256.314,E2 -256.314} C_VEL
